   // GBK_TO_UNICODE[32068] := 16#DCDB;
   // GBK_TO_UNICODE[32069] := 16#82D2;
   // GBK_TO_UNICODE[32070] := 16#DCDC;
   // GBK_TO_UNICODE[32071] := 16#82D8;
   // GBK_TO_UNICODE[32072] := 16#DCDD;
   // GBK_TO_UNICODE[32073] := 16#830C;
   // GBK_TO_UNICODE[32074] := 16#DCDE;
   // GBK_TO_UNICODE[32075] := 16#82FB;
   // GBK_TO_UNICODE[32076] := 16#DCDF;
   // GBK_TO_UNICODE[32077] := 16#82D3;
   // GBK_TO_UNICODE[32078] := 16#DCE0;
   // GBK_TO_UNICODE[32079] := 16#8311;
   // GBK_TO_UNICODE[32080] := 16#DCE1;
   // GBK_TO_UNICODE[32081] := 16#831A;
   // GBK_TO_UNICODE[32082] := 16#DCE2;
   // GBK_TO_UNICODE[32083] := 16#8306;
   // GBK_TO_UNICODE[32084] := 16#DCE3;
   // GBK_TO_UNICODE[32085] := 16#8314;
   // GBK_TO_UNICODE[32086] := 16#DCE4;
   // GBK_TO_UNICODE[32087] := 16#8315;
   // GBK_TO_UNICODE[32088] := 16#DCE5;
   // GBK_TO_UNICODE[32089] := 16#82E0;
   // GBK_TO_UNICODE[32090] := 16#DCE6;
   // GBK_TO_UNICODE[32091] := 16#82D5;
   // GBK_TO_UNICODE[32092] := 16#DCE7;
   // GBK_TO_UNICODE[32093] := 16#831C;
   // GBK_TO_UNICODE[32094] := 16#DCE8;
   // GBK_TO_UNICODE[32095] := 16#8351;
   // GBK_TO_UNICODE[32096] := 16#DCE9;
   // GBK_TO_UNICODE[32097] := 16#835B;
   // GBK_TO_UNICODE[32098] := 16#DCEA;
   // GBK_TO_UNICODE[32099] := 16#835C;
   // GBK_TO_UNICODE[32100] := 16#DCEB;
   // GBK_TO_UNICODE[32101] := 16#8308;
   // GBK_TO_UNICODE[32102] := 16#DCEC;
   // GBK_TO_UNICODE[32103] := 16#8392;
   // GBK_TO_UNICODE[32104] := 16#DCED;
   // GBK_TO_UNICODE[32105] := 16#833C;
   // GBK_TO_UNICODE[32106] := 16#DCEE;
   // GBK_TO_UNICODE[32107] := 16#8334;
   // GBK_TO_UNICODE[32108] := 16#DCEF;
   // GBK_TO_UNICODE[32109] := 16#8331;
   // GBK_TO_UNICODE[32110] := 16#DCF0;
   // GBK_TO_UNICODE[32111] := 16#839B;
   // GBK_TO_UNICODE[32112] := 16#DCF1;
   // GBK_TO_UNICODE[32113] := 16#835E;
   // GBK_TO_UNICODE[32114] := 16#DCF2;
   // GBK_TO_UNICODE[32115] := 16#832F;
   // GBK_TO_UNICODE[32116] := 16#DCF3;
   // GBK_TO_UNICODE[32117] := 16#834F;
   // GBK_TO_UNICODE[32118] := 16#DCF4;
   // GBK_TO_UNICODE[32119] := 16#8347;
   // GBK_TO_UNICODE[32120] := 16#DCF5;
   // GBK_TO_UNICODE[32121] := 16#8343;
   // GBK_TO_UNICODE[32122] := 16#DCF6;
   // GBK_TO_UNICODE[32123] := 16#835F;
   // GBK_TO_UNICODE[32124] := 16#DCF7;
   // GBK_TO_UNICODE[32125] := 16#8340;
   // GBK_TO_UNICODE[32126] := 16#DCF8;
   // GBK_TO_UNICODE[32127] := 16#8317;
   // GBK_TO_UNICODE[32128] := 16#DCF9;
   // GBK_TO_UNICODE[32129] := 16#8360;
   // GBK_TO_UNICODE[32130] := 16#DCFA;
   // GBK_TO_UNICODE[32131] := 16#832D;
   // GBK_TO_UNICODE[32132] := 16#DCFB;
   // GBK_TO_UNICODE[32133] := 16#833A;
   // GBK_TO_UNICODE[32134] := 16#DCFC;
   // GBK_TO_UNICODE[32135] := 16#8333;
   // GBK_TO_UNICODE[32136] := 16#DCFD;
   // GBK_TO_UNICODE[32137] := 16#8366;
   // GBK_TO_UNICODE[32138] := 16#DCFE;
   // GBK_TO_UNICODE[32139] := 16#8365;
   // GBK_TO_UNICODE[32140] := 16#DD40;
   // GBK_TO_UNICODE[32141] := 16#8EE5;
   // GBK_TO_UNICODE[32142] := 16#DD41;
   // GBK_TO_UNICODE[32143] := 16#8EE6;
   // GBK_TO_UNICODE[32144] := 16#DD42;
   // GBK_TO_UNICODE[32145] := 16#8EE7;
   // GBK_TO_UNICODE[32146] := 16#DD43;
   // GBK_TO_UNICODE[32147] := 16#8EE8;
   // GBK_TO_UNICODE[32148] := 16#DD44;
   // GBK_TO_UNICODE[32149] := 16#8EE9;
   // GBK_TO_UNICODE[32150] := 16#DD45;
   // GBK_TO_UNICODE[32151] := 16#8EEA;
   // GBK_TO_UNICODE[32152] := 16#DD46;
   // GBK_TO_UNICODE[32153] := 16#8EEB;
   // GBK_TO_UNICODE[32154] := 16#DD47;
   // GBK_TO_UNICODE[32155] := 16#8EEC;
   // GBK_TO_UNICODE[32156] := 16#DD48;
   // GBK_TO_UNICODE[32157] := 16#8EED;
   // GBK_TO_UNICODE[32158] := 16#DD49;
   // GBK_TO_UNICODE[32159] := 16#8EEE;
   // GBK_TO_UNICODE[32160] := 16#DD4A;
   // GBK_TO_UNICODE[32161] := 16#8EEF;
   // GBK_TO_UNICODE[32162] := 16#DD4B;
   // GBK_TO_UNICODE[32163] := 16#8EF0;
   // GBK_TO_UNICODE[32164] := 16#DD4C;
   // GBK_TO_UNICODE[32165] := 16#8EF1;
   // GBK_TO_UNICODE[32166] := 16#DD4D;
   // GBK_TO_UNICODE[32167] := 16#8EF2;
   // GBK_TO_UNICODE[32168] := 16#DD4E;
   // GBK_TO_UNICODE[32169] := 16#8EF3;
   // GBK_TO_UNICODE[32170] := 16#DD4F;
   // GBK_TO_UNICODE[32171] := 16#8EF4;
   // GBK_TO_UNICODE[32172] := 16#DD50;
   // GBK_TO_UNICODE[32173] := 16#8EF5;
   // GBK_TO_UNICODE[32174] := 16#DD51;
   // GBK_TO_UNICODE[32175] := 16#8EF6;
   // GBK_TO_UNICODE[32176] := 16#DD52;
   // GBK_TO_UNICODE[32177] := 16#8EF7;
   // GBK_TO_UNICODE[32178] := 16#DD53;
   // GBK_TO_UNICODE[32179] := 16#8EF8;
   // GBK_TO_UNICODE[32180] := 16#DD54;
   // GBK_TO_UNICODE[32181] := 16#8EF9;
   // GBK_TO_UNICODE[32182] := 16#DD55;
   // GBK_TO_UNICODE[32183] := 16#8EFA;
   // GBK_TO_UNICODE[32184] := 16#DD56;
   // GBK_TO_UNICODE[32185] := 16#8EFB;
   // GBK_TO_UNICODE[32186] := 16#DD57;
   // GBK_TO_UNICODE[32187] := 16#8EFC;
   // GBK_TO_UNICODE[32188] := 16#DD58;
   // GBK_TO_UNICODE[32189] := 16#8EFD;
   // GBK_TO_UNICODE[32190] := 16#DD59;
   // GBK_TO_UNICODE[32191] := 16#8EFE;
   // GBK_TO_UNICODE[32192] := 16#DD5A;
   // GBK_TO_UNICODE[32193] := 16#8EFF;
   // GBK_TO_UNICODE[32194] := 16#DD5B;
   // GBK_TO_UNICODE[32195] := 16#8F00;
   // GBK_TO_UNICODE[32196] := 16#DD5C;
   // GBK_TO_UNICODE[32197] := 16#8F01;
   // GBK_TO_UNICODE[32198] := 16#DD5D;
   // GBK_TO_UNICODE[32199] := 16#8F02;
   // GBK_TO_UNICODE[32200] := 16#DD5E;
   // GBK_TO_UNICODE[32201] := 16#8F03;
   // GBK_TO_UNICODE[32202] := 16#DD5F;
   // GBK_TO_UNICODE[32203] := 16#8F04;
   // GBK_TO_UNICODE[32204] := 16#DD60;
   // GBK_TO_UNICODE[32205] := 16#8F05;
   // GBK_TO_UNICODE[32206] := 16#DD61;
   // GBK_TO_UNICODE[32207] := 16#8F06;
   // GBK_TO_UNICODE[32208] := 16#DD62;
   // GBK_TO_UNICODE[32209] := 16#8F07;
   // GBK_TO_UNICODE[32210] := 16#DD63;
   // GBK_TO_UNICODE[32211] := 16#8F08;
   // GBK_TO_UNICODE[32212] := 16#DD64;
   // GBK_TO_UNICODE[32213] := 16#8F09;
   // GBK_TO_UNICODE[32214] := 16#DD65;
   // GBK_TO_UNICODE[32215] := 16#8F0A;
   // GBK_TO_UNICODE[32216] := 16#DD66;
   // GBK_TO_UNICODE[32217] := 16#8F0B;
   // GBK_TO_UNICODE[32218] := 16#DD67;
   // GBK_TO_UNICODE[32219] := 16#8F0C;
   // GBK_TO_UNICODE[32220] := 16#DD68;
   // GBK_TO_UNICODE[32221] := 16#8F0D;
   // GBK_TO_UNICODE[32222] := 16#DD69;
   // GBK_TO_UNICODE[32223] := 16#8F0E;
   // GBK_TO_UNICODE[32224] := 16#DD6A;
   // GBK_TO_UNICODE[32225] := 16#8F0F;
   // GBK_TO_UNICODE[32226] := 16#DD6B;
   // GBK_TO_UNICODE[32227] := 16#8F10;
   // GBK_TO_UNICODE[32228] := 16#DD6C;
   // GBK_TO_UNICODE[32229] := 16#8F11;
   // GBK_TO_UNICODE[32230] := 16#DD6D;
   // GBK_TO_UNICODE[32231] := 16#8F12;
   // GBK_TO_UNICODE[32232] := 16#DD6E;
   // GBK_TO_UNICODE[32233] := 16#8F13;
   // GBK_TO_UNICODE[32234] := 16#DD6F;
   // GBK_TO_UNICODE[32235] := 16#8F14;
   // GBK_TO_UNICODE[32236] := 16#DD70;
   // GBK_TO_UNICODE[32237] := 16#8F15;
   // GBK_TO_UNICODE[32238] := 16#DD71;
   // GBK_TO_UNICODE[32239] := 16#8F16;
   // GBK_TO_UNICODE[32240] := 16#DD72;
   // GBK_TO_UNICODE[32241] := 16#8F17;
   // GBK_TO_UNICODE[32242] := 16#DD73;
   // GBK_TO_UNICODE[32243] := 16#8F18;
   // GBK_TO_UNICODE[32244] := 16#DD74;
   // GBK_TO_UNICODE[32245] := 16#8F19;
   // GBK_TO_UNICODE[32246] := 16#DD75;
   // GBK_TO_UNICODE[32247] := 16#8F1A;
   // GBK_TO_UNICODE[32248] := 16#DD76;
   // GBK_TO_UNICODE[32249] := 16#8F1B;
   // GBK_TO_UNICODE[32250] := 16#DD77;
   // GBK_TO_UNICODE[32251] := 16#8F1C;
   // GBK_TO_UNICODE[32252] := 16#DD78;
   // GBK_TO_UNICODE[32253] := 16#8F1D;
   // GBK_TO_UNICODE[32254] := 16#DD79;
   // GBK_TO_UNICODE[32255] := 16#8F1E;
   // GBK_TO_UNICODE[32256] := 16#DD7A;
   // GBK_TO_UNICODE[32257] := 16#8F1F;
   // GBK_TO_UNICODE[32258] := 16#DD7B;
   // GBK_TO_UNICODE[32259] := 16#8F20;
   // GBK_TO_UNICODE[32260] := 16#DD7C;
   // GBK_TO_UNICODE[32261] := 16#8F21;
   // GBK_TO_UNICODE[32262] := 16#DD7D;
   // GBK_TO_UNICODE[32263] := 16#8F22;
   // GBK_TO_UNICODE[32264] := 16#DD7E;
   // GBK_TO_UNICODE[32265] := 16#8F23;
   // GBK_TO_UNICODE[32266] := 16#DD80;
   // GBK_TO_UNICODE[32267] := 16#8F24;
   // GBK_TO_UNICODE[32268] := 16#DD81;
   // GBK_TO_UNICODE[32269] := 16#8F25;
   // GBK_TO_UNICODE[32270] := 16#DD82;
   // GBK_TO_UNICODE[32271] := 16#8F26;
   // GBK_TO_UNICODE[32272] := 16#DD83;
   // GBK_TO_UNICODE[32273] := 16#8F27;
   // GBK_TO_UNICODE[32274] := 16#DD84;
   // GBK_TO_UNICODE[32275] := 16#8F28;
   // GBK_TO_UNICODE[32276] := 16#DD85;
   // GBK_TO_UNICODE[32277] := 16#8F29;
   // GBK_TO_UNICODE[32278] := 16#DD86;
   // GBK_TO_UNICODE[32279] := 16#8F2A;
   // GBK_TO_UNICODE[32280] := 16#DD87;
   // GBK_TO_UNICODE[32281] := 16#8F2B;
   // GBK_TO_UNICODE[32282] := 16#DD88;
   // GBK_TO_UNICODE[32283] := 16#8F2C;
   // GBK_TO_UNICODE[32284] := 16#DD89;
   // GBK_TO_UNICODE[32285] := 16#8F2D;
   // GBK_TO_UNICODE[32286] := 16#DD8A;
   // GBK_TO_UNICODE[32287] := 16#8F2E;
   // GBK_TO_UNICODE[32288] := 16#DD8B;
   // GBK_TO_UNICODE[32289] := 16#8F2F;
   // GBK_TO_UNICODE[32290] := 16#DD8C;
   // GBK_TO_UNICODE[32291] := 16#8F30;
   // GBK_TO_UNICODE[32292] := 16#DD8D;
   // GBK_TO_UNICODE[32293] := 16#8F31;
   // GBK_TO_UNICODE[32294] := 16#DD8E;
   // GBK_TO_UNICODE[32295] := 16#8F32;
   // GBK_TO_UNICODE[32296] := 16#DD8F;
   // GBK_TO_UNICODE[32297] := 16#8F33;
   // GBK_TO_UNICODE[32298] := 16#DD90;
   // GBK_TO_UNICODE[32299] := 16#8F34;
   // GBK_TO_UNICODE[32300] := 16#DD91;
   // GBK_TO_UNICODE[32301] := 16#8F35;
   // GBK_TO_UNICODE[32302] := 16#DD92;
   // GBK_TO_UNICODE[32303] := 16#8F36;
   // GBK_TO_UNICODE[32304] := 16#DD93;
   // GBK_TO_UNICODE[32305] := 16#8F37;
   // GBK_TO_UNICODE[32306] := 16#DD94;
   // GBK_TO_UNICODE[32307] := 16#8F38;
   // GBK_TO_UNICODE[32308] := 16#DD95;
   // GBK_TO_UNICODE[32309] := 16#8F39;
   // GBK_TO_UNICODE[32310] := 16#DD96;
   // GBK_TO_UNICODE[32311] := 16#8F3A;
   // GBK_TO_UNICODE[32312] := 16#DD97;
   // GBK_TO_UNICODE[32313] := 16#8F3B;
   // GBK_TO_UNICODE[32314] := 16#DD98;
   // GBK_TO_UNICODE[32315] := 16#8F3C;
   // GBK_TO_UNICODE[32316] := 16#DD99;
   // GBK_TO_UNICODE[32317] := 16#8F3D;
   // GBK_TO_UNICODE[32318] := 16#DD9A;
   // GBK_TO_UNICODE[32319] := 16#8F3E;
   // GBK_TO_UNICODE[32320] := 16#DD9B;
   // GBK_TO_UNICODE[32321] := 16#8F3F;
   // GBK_TO_UNICODE[32322] := 16#DD9C;
   // GBK_TO_UNICODE[32323] := 16#8F40;
   // GBK_TO_UNICODE[32324] := 16#DD9D;
   // GBK_TO_UNICODE[32325] := 16#8F41;
   // GBK_TO_UNICODE[32326] := 16#DD9E;
   // GBK_TO_UNICODE[32327] := 16#8F42;
   // GBK_TO_UNICODE[32328] := 16#DD9F;
   // GBK_TO_UNICODE[32329] := 16#8F43;
   // GBK_TO_UNICODE[32330] := 16#DDA0;
   // GBK_TO_UNICODE[32331] := 16#8F44;
   // GBK_TO_UNICODE[32332] := 16#DDA1;
   // GBK_TO_UNICODE[32333] := 16#8368;
   // GBK_TO_UNICODE[32334] := 16#DDA2;
   // GBK_TO_UNICODE[32335] := 16#831B;
   // GBK_TO_UNICODE[32336] := 16#DDA3;
   // GBK_TO_UNICODE[32337] := 16#8369;
   // GBK_TO_UNICODE[32338] := 16#DDA4;
   // GBK_TO_UNICODE[32339] := 16#836C;
   // GBK_TO_UNICODE[32340] := 16#DDA5;
   // GBK_TO_UNICODE[32341] := 16#836A;
   // GBK_TO_UNICODE[32342] := 16#DDA6;
   // GBK_TO_UNICODE[32343] := 16#836D;
   // GBK_TO_UNICODE[32344] := 16#DDA7;
   // GBK_TO_UNICODE[32345] := 16#836E;
   // GBK_TO_UNICODE[32346] := 16#DDA8;
   // GBK_TO_UNICODE[32347] := 16#83B0;
   // GBK_TO_UNICODE[32348] := 16#DDA9;
   // GBK_TO_UNICODE[32349] := 16#8378;
   // GBK_TO_UNICODE[32350] := 16#DDAA;
   // GBK_TO_UNICODE[32351] := 16#83B3;
   // GBK_TO_UNICODE[32352] := 16#DDAB;
   // GBK_TO_UNICODE[32353] := 16#83B4;
   // GBK_TO_UNICODE[32354] := 16#DDAC;
   // GBK_TO_UNICODE[32355] := 16#83A0;
   // GBK_TO_UNICODE[32356] := 16#DDAD;
   // GBK_TO_UNICODE[32357] := 16#83AA;
   // GBK_TO_UNICODE[32358] := 16#DDAE;
   // GBK_TO_UNICODE[32359] := 16#8393;
   // GBK_TO_UNICODE[32360] := 16#DDAF;
   // GBK_TO_UNICODE[32361] := 16#839C;
   // GBK_TO_UNICODE[32362] := 16#DDB0;
   // GBK_TO_UNICODE[32363] := 16#8385;
   // GBK_TO_UNICODE[32364] := 16#DDB1;
   // GBK_TO_UNICODE[32365] := 16#837C;
   // GBK_TO_UNICODE[32366] := 16#DDB2;
   // GBK_TO_UNICODE[32367] := 16#83B6;
   // GBK_TO_UNICODE[32368] := 16#DDB3;
   // GBK_TO_UNICODE[32369] := 16#83A9;
   // GBK_TO_UNICODE[32370] := 16#DDB4;
   // GBK_TO_UNICODE[32371] := 16#837D;
   // GBK_TO_UNICODE[32372] := 16#DDB5;
   // GBK_TO_UNICODE[32373] := 16#83B8;
   // GBK_TO_UNICODE[32374] := 16#DDB6;
   // GBK_TO_UNICODE[32375] := 16#837B;
   // GBK_TO_UNICODE[32376] := 16#DDB7;
   // GBK_TO_UNICODE[32377] := 16#8398;
   // GBK_TO_UNICODE[32378] := 16#DDB8;
   // GBK_TO_UNICODE[32379] := 16#839E;
   // GBK_TO_UNICODE[32380] := 16#DDB9;
   // GBK_TO_UNICODE[32381] := 16#83A8;
   // GBK_TO_UNICODE[32382] := 16#DDBA;
   // GBK_TO_UNICODE[32383] := 16#83BA;
   // GBK_TO_UNICODE[32384] := 16#DDBB;
   // GBK_TO_UNICODE[32385] := 16#83BC;
   // GBK_TO_UNICODE[32386] := 16#DDBC;
   // GBK_TO_UNICODE[32387] := 16#83C1;
   // GBK_TO_UNICODE[32388] := 16#DDBD;
   // GBK_TO_UNICODE[32389] := 16#8401;
   // GBK_TO_UNICODE[32390] := 16#DDBE;
   // GBK_TO_UNICODE[32391] := 16#83E5;
   // GBK_TO_UNICODE[32392] := 16#DDBF;
   // GBK_TO_UNICODE[32393] := 16#83D8;
   // GBK_TO_UNICODE[32394] := 16#DDC0;
   // GBK_TO_UNICODE[32395] := 16#5807;
   // GBK_TO_UNICODE[32396] := 16#DDC1;
   // GBK_TO_UNICODE[32397] := 16#8418;
   // GBK_TO_UNICODE[32398] := 16#DDC2;
   // GBK_TO_UNICODE[32399] := 16#840B;
   // GBK_TO_UNICODE[32400] := 16#DDC3;
   // GBK_TO_UNICODE[32401] := 16#83DD;
   // GBK_TO_UNICODE[32402] := 16#DDC4;
   // GBK_TO_UNICODE[32403] := 16#83FD;
   // GBK_TO_UNICODE[32404] := 16#DDC5;
   // GBK_TO_UNICODE[32405] := 16#83D6;
   // GBK_TO_UNICODE[32406] := 16#DDC6;
   // GBK_TO_UNICODE[32407] := 16#841C;
   // GBK_TO_UNICODE[32408] := 16#DDC7;
   // GBK_TO_UNICODE[32409] := 16#8438;
   // GBK_TO_UNICODE[32410] := 16#DDC8;
   // GBK_TO_UNICODE[32411] := 16#8411;
   // GBK_TO_UNICODE[32412] := 16#DDC9;
   // GBK_TO_UNICODE[32413] := 16#8406;
   // GBK_TO_UNICODE[32414] := 16#DDCA;
   // GBK_TO_UNICODE[32415] := 16#83D4;
   // GBK_TO_UNICODE[32416] := 16#DDCB;
   // GBK_TO_UNICODE[32417] := 16#83DF;
   // GBK_TO_UNICODE[32418] := 16#DDCC;
   // GBK_TO_UNICODE[32419] := 16#840F;
   // GBK_TO_UNICODE[32420] := 16#DDCD;
   // GBK_TO_UNICODE[32421] := 16#8403;
   // GBK_TO_UNICODE[32422] := 16#DDCE;
   // GBK_TO_UNICODE[32423] := 16#83F8;
   // GBK_TO_UNICODE[32424] := 16#DDCF;
   // GBK_TO_UNICODE[32425] := 16#83F9;
   // GBK_TO_UNICODE[32426] := 16#DDD0;
   // GBK_TO_UNICODE[32427] := 16#83EA;
   // GBK_TO_UNICODE[32428] := 16#DDD1;
   // GBK_TO_UNICODE[32429] := 16#83C5;
   // GBK_TO_UNICODE[32430] := 16#DDD2;
   // GBK_TO_UNICODE[32431] := 16#83C0;
   // GBK_TO_UNICODE[32432] := 16#DDD3;
   // GBK_TO_UNICODE[32433] := 16#8426;
   // GBK_TO_UNICODE[32434] := 16#DDD4;
   // GBK_TO_UNICODE[32435] := 16#83F0;
   // GBK_TO_UNICODE[32436] := 16#DDD5;
   // GBK_TO_UNICODE[32437] := 16#83E1;
   // GBK_TO_UNICODE[32438] := 16#DDD6;
   // GBK_TO_UNICODE[32439] := 16#845C;
   // GBK_TO_UNICODE[32440] := 16#DDD7;
   // GBK_TO_UNICODE[32441] := 16#8451;
   // GBK_TO_UNICODE[32442] := 16#DDD8;
   // GBK_TO_UNICODE[32443] := 16#845A;
   // GBK_TO_UNICODE[32444] := 16#DDD9;
   // GBK_TO_UNICODE[32445] := 16#8459;
   // GBK_TO_UNICODE[32446] := 16#DDDA;
   // GBK_TO_UNICODE[32447] := 16#8473;
   // GBK_TO_UNICODE[32448] := 16#DDDB;
   // GBK_TO_UNICODE[32449] := 16#8487;
   // GBK_TO_UNICODE[32450] := 16#DDDC;
   // GBK_TO_UNICODE[32451] := 16#8488;
   // GBK_TO_UNICODE[32452] := 16#DDDD;
   // GBK_TO_UNICODE[32453] := 16#847A;
   // GBK_TO_UNICODE[32454] := 16#DDDE;
   // GBK_TO_UNICODE[32455] := 16#8489;
   // GBK_TO_UNICODE[32456] := 16#DDDF;
   // GBK_TO_UNICODE[32457] := 16#8478;
   // GBK_TO_UNICODE[32458] := 16#DDE0;
   // GBK_TO_UNICODE[32459] := 16#843C;
   // GBK_TO_UNICODE[32460] := 16#DDE1;
   // GBK_TO_UNICODE[32461] := 16#8446;
   // GBK_TO_UNICODE[32462] := 16#DDE2;
   // GBK_TO_UNICODE[32463] := 16#8469;
   // GBK_TO_UNICODE[32464] := 16#DDE3;
   // GBK_TO_UNICODE[32465] := 16#8476;
   // GBK_TO_UNICODE[32466] := 16#DDE4;
   // GBK_TO_UNICODE[32467] := 16#848C;
   // GBK_TO_UNICODE[32468] := 16#DDE5;
   // GBK_TO_UNICODE[32469] := 16#848E;
   // GBK_TO_UNICODE[32470] := 16#DDE6;
   // GBK_TO_UNICODE[32471] := 16#8431;
   // GBK_TO_UNICODE[32472] := 16#DDE7;
   // GBK_TO_UNICODE[32473] := 16#846D;
   // GBK_TO_UNICODE[32474] := 16#DDE8;
   // GBK_TO_UNICODE[32475] := 16#84C1;
   // GBK_TO_UNICODE[32476] := 16#DDE9;
   // GBK_TO_UNICODE[32477] := 16#84CD;
   // GBK_TO_UNICODE[32478] := 16#DDEA;
   // GBK_TO_UNICODE[32479] := 16#84D0;
   // GBK_TO_UNICODE[32480] := 16#DDEB;
   // GBK_TO_UNICODE[32481] := 16#84E6;
   // GBK_TO_UNICODE[32482] := 16#DDEC;
   // GBK_TO_UNICODE[32483] := 16#84BD;
   // GBK_TO_UNICODE[32484] := 16#DDED;
   // GBK_TO_UNICODE[32485] := 16#84D3;
   // GBK_TO_UNICODE[32486] := 16#DDEE;
   // GBK_TO_UNICODE[32487] := 16#84CA;
   // GBK_TO_UNICODE[32488] := 16#DDEF;
   // GBK_TO_UNICODE[32489] := 16#84BF;
   // GBK_TO_UNICODE[32490] := 16#DDF0;
   // GBK_TO_UNICODE[32491] := 16#84BA;
   // GBK_TO_UNICODE[32492] := 16#DDF1;
   // GBK_TO_UNICODE[32493] := 16#84E0;
   // GBK_TO_UNICODE[32494] := 16#DDF2;
   // GBK_TO_UNICODE[32495] := 16#84A1;
   // GBK_TO_UNICODE[32496] := 16#DDF3;
   // GBK_TO_UNICODE[32497] := 16#84B9;
   // GBK_TO_UNICODE[32498] := 16#DDF4;
   // GBK_TO_UNICODE[32499] := 16#84B4;
   // GBK_TO_UNICODE[32500] := 16#DDF5;
   // GBK_TO_UNICODE[32501] := 16#8497;
   // GBK_TO_UNICODE[32502] := 16#DDF6;
   // GBK_TO_UNICODE[32503] := 16#84E5;
   // GBK_TO_UNICODE[32504] := 16#DDF7;
   // GBK_TO_UNICODE[32505] := 16#84E3;
   // GBK_TO_UNICODE[32506] := 16#DDF8;
   // GBK_TO_UNICODE[32507] := 16#850C;
   // GBK_TO_UNICODE[32508] := 16#DDF9;
   // GBK_TO_UNICODE[32509] := 16#750D;
   // GBK_TO_UNICODE[32510] := 16#DDFA;
   // GBK_TO_UNICODE[32511] := 16#8538;
   // GBK_TO_UNICODE[32512] := 16#DDFB;
   // GBK_TO_UNICODE[32513] := 16#84F0;
   // GBK_TO_UNICODE[32514] := 16#DDFC;
   // GBK_TO_UNICODE[32515] := 16#8539;
   // GBK_TO_UNICODE[32516] := 16#DDFD;
   // GBK_TO_UNICODE[32517] := 16#851F;
   // GBK_TO_UNICODE[32518] := 16#DDFE;
   // GBK_TO_UNICODE[32519] := 16#853A;
   // GBK_TO_UNICODE[32520] := 16#DE40;
   // GBK_TO_UNICODE[32521] := 16#8F45;
   // GBK_TO_UNICODE[32522] := 16#DE41;
   // GBK_TO_UNICODE[32523] := 16#8F46;
   // GBK_TO_UNICODE[32524] := 16#DE42;
   // GBK_TO_UNICODE[32525] := 16#8F47;
   // GBK_TO_UNICODE[32526] := 16#DE43;
   // GBK_TO_UNICODE[32527] := 16#8F48;
   // GBK_TO_UNICODE[32528] := 16#DE44;
   // GBK_TO_UNICODE[32529] := 16#8F49;
   // GBK_TO_UNICODE[32530] := 16#DE45;
   // GBK_TO_UNICODE[32531] := 16#8F4A;
   // GBK_TO_UNICODE[32532] := 16#DE46;
   // GBK_TO_UNICODE[32533] := 16#8F4B;
   // GBK_TO_UNICODE[32534] := 16#DE47;
   // GBK_TO_UNICODE[32535] := 16#8F4C;
   // GBK_TO_UNICODE[32536] := 16#DE48;
   // GBK_TO_UNICODE[32537] := 16#8F4D;
   // GBK_TO_UNICODE[32538] := 16#DE49;
   // GBK_TO_UNICODE[32539] := 16#8F4E;
   // GBK_TO_UNICODE[32540] := 16#DE4A;
   // GBK_TO_UNICODE[32541] := 16#8F4F;
   // GBK_TO_UNICODE[32542] := 16#DE4B;
   // GBK_TO_UNICODE[32543] := 16#8F50;
   // GBK_TO_UNICODE[32544] := 16#DE4C;
   // GBK_TO_UNICODE[32545] := 16#8F51;
   // GBK_TO_UNICODE[32546] := 16#DE4D;
   // GBK_TO_UNICODE[32547] := 16#8F52;
   // GBK_TO_UNICODE[32548] := 16#DE4E;
   // GBK_TO_UNICODE[32549] := 16#8F53;
   // GBK_TO_UNICODE[32550] := 16#DE4F;
   // GBK_TO_UNICODE[32551] := 16#8F54;
   // GBK_TO_UNICODE[32552] := 16#DE50;
   // GBK_TO_UNICODE[32553] := 16#8F55;
   // GBK_TO_UNICODE[32554] := 16#DE51;
   // GBK_TO_UNICODE[32555] := 16#8F56;
   // GBK_TO_UNICODE[32556] := 16#DE52;
   // GBK_TO_UNICODE[32557] := 16#8F57;
   // GBK_TO_UNICODE[32558] := 16#DE53;
   // GBK_TO_UNICODE[32559] := 16#8F58;
   // GBK_TO_UNICODE[32560] := 16#DE54;
   // GBK_TO_UNICODE[32561] := 16#8F59;
   // GBK_TO_UNICODE[32562] := 16#DE55;
   // GBK_TO_UNICODE[32563] := 16#8F5A;
   // GBK_TO_UNICODE[32564] := 16#DE56;
   // GBK_TO_UNICODE[32565] := 16#8F5B;
   // GBK_TO_UNICODE[32566] := 16#DE57;
   // GBK_TO_UNICODE[32567] := 16#8F5C;
   // GBK_TO_UNICODE[32568] := 16#DE58;
   // GBK_TO_UNICODE[32569] := 16#8F5D;
   // GBK_TO_UNICODE[32570] := 16#DE59;
   // GBK_TO_UNICODE[32571] := 16#8F5E;
   // GBK_TO_UNICODE[32572] := 16#DE5A;
   // GBK_TO_UNICODE[32573] := 16#8F5F;
   // GBK_TO_UNICODE[32574] := 16#DE5B;
   // GBK_TO_UNICODE[32575] := 16#8F60;
   // GBK_TO_UNICODE[32576] := 16#DE5C;
   // GBK_TO_UNICODE[32577] := 16#8F61;
   // GBK_TO_UNICODE[32578] := 16#DE5D;
   // GBK_TO_UNICODE[32579] := 16#8F62;
   // GBK_TO_UNICODE[32580] := 16#DE5E;
   // GBK_TO_UNICODE[32581] := 16#8F63;
   // GBK_TO_UNICODE[32582] := 16#DE5F;
   // GBK_TO_UNICODE[32583] := 16#8F64;
   // GBK_TO_UNICODE[32584] := 16#DE60;
   // GBK_TO_UNICODE[32585] := 16#8F65;
   // GBK_TO_UNICODE[32586] := 16#DE61;
   // GBK_TO_UNICODE[32587] := 16#8F6A;
   // GBK_TO_UNICODE[32588] := 16#DE62;
   // GBK_TO_UNICODE[32589] := 16#8F80;
   // GBK_TO_UNICODE[32590] := 16#DE63;
   // GBK_TO_UNICODE[32591] := 16#8F8C;
   // GBK_TO_UNICODE[32592] := 16#DE64;
   // GBK_TO_UNICODE[32593] := 16#8F92;
   // GBK_TO_UNICODE[32594] := 16#DE65;
   // GBK_TO_UNICODE[32595] := 16#8F9D;
   // GBK_TO_UNICODE[32596] := 16#DE66;
   // GBK_TO_UNICODE[32597] := 16#8FA0;
   // GBK_TO_UNICODE[32598] := 16#DE67;
   // GBK_TO_UNICODE[32599] := 16#8FA1;
   // GBK_TO_UNICODE[32600] := 16#DE68;
   // GBK_TO_UNICODE[32601] := 16#8FA2;
   // GBK_TO_UNICODE[32602] := 16#DE69;
   // GBK_TO_UNICODE[32603] := 16#8FA4;
   // GBK_TO_UNICODE[32604] := 16#DE6A;
   // GBK_TO_UNICODE[32605] := 16#8FA5;
   // GBK_TO_UNICODE[32606] := 16#DE6B;
   // GBK_TO_UNICODE[32607] := 16#8FA6;
   // GBK_TO_UNICODE[32608] := 16#DE6C;
   // GBK_TO_UNICODE[32609] := 16#8FA7;
   // GBK_TO_UNICODE[32610] := 16#DE6D;
   // GBK_TO_UNICODE[32611] := 16#8FAA;
   // GBK_TO_UNICODE[32612] := 16#DE6E;
   // GBK_TO_UNICODE[32613] := 16#8FAC;
   // GBK_TO_UNICODE[32614] := 16#DE6F;
   // GBK_TO_UNICODE[32615] := 16#8FAD;
   // GBK_TO_UNICODE[32616] := 16#DE70;
   // GBK_TO_UNICODE[32617] := 16#8FAE;
   // GBK_TO_UNICODE[32618] := 16#DE71;
   // GBK_TO_UNICODE[32619] := 16#8FAF;
   // GBK_TO_UNICODE[32620] := 16#DE72;
   // GBK_TO_UNICODE[32621] := 16#8FB2;
   // GBK_TO_UNICODE[32622] := 16#DE73;
   // GBK_TO_UNICODE[32623] := 16#8FB3;
   // GBK_TO_UNICODE[32624] := 16#DE74;
   // GBK_TO_UNICODE[32625] := 16#8FB4;
   // GBK_TO_UNICODE[32626] := 16#DE75;
   // GBK_TO_UNICODE[32627] := 16#8FB5;
   // GBK_TO_UNICODE[32628] := 16#DE76;
   // GBK_TO_UNICODE[32629] := 16#8FB7;
   // GBK_TO_UNICODE[32630] := 16#DE77;
   // GBK_TO_UNICODE[32631] := 16#8FB8;
   // GBK_TO_UNICODE[32632] := 16#DE78;
   // GBK_TO_UNICODE[32633] := 16#8FBA;
   // GBK_TO_UNICODE[32634] := 16#DE79;
   // GBK_TO_UNICODE[32635] := 16#8FBB;
   // GBK_TO_UNICODE[32636] := 16#DE7A;
   // GBK_TO_UNICODE[32637] := 16#8FBC;
   // GBK_TO_UNICODE[32638] := 16#DE7B;
   // GBK_TO_UNICODE[32639] := 16#8FBF;
   // GBK_TO_UNICODE[32640] := 16#DE7C;
   // GBK_TO_UNICODE[32641] := 16#8FC0;
   // GBK_TO_UNICODE[32642] := 16#DE7D;
   // GBK_TO_UNICODE[32643] := 16#8FC3;
   // GBK_TO_UNICODE[32644] := 16#DE7E;
   // GBK_TO_UNICODE[32645] := 16#8FC6;
   // GBK_TO_UNICODE[32646] := 16#DE80;
   // GBK_TO_UNICODE[32647] := 16#8FC9;
   // GBK_TO_UNICODE[32648] := 16#DE81;
   // GBK_TO_UNICODE[32649] := 16#8FCA;
   // GBK_TO_UNICODE[32650] := 16#DE82;
   // GBK_TO_UNICODE[32651] := 16#8FCB;
   // GBK_TO_UNICODE[32652] := 16#DE83;
   // GBK_TO_UNICODE[32653] := 16#8FCC;
   // GBK_TO_UNICODE[32654] := 16#DE84;
   // GBK_TO_UNICODE[32655] := 16#8FCD;
   // GBK_TO_UNICODE[32656] := 16#DE85;
   // GBK_TO_UNICODE[32657] := 16#8FCF;
   // GBK_TO_UNICODE[32658] := 16#DE86;
   // GBK_TO_UNICODE[32659] := 16#8FD2;
   // GBK_TO_UNICODE[32660] := 16#DE87;
   // GBK_TO_UNICODE[32661] := 16#8FD6;
   // GBK_TO_UNICODE[32662] := 16#DE88;
   // GBK_TO_UNICODE[32663] := 16#8FD7;
   // GBK_TO_UNICODE[32664] := 16#DE89;
   // GBK_TO_UNICODE[32665] := 16#8FDA;
   // GBK_TO_UNICODE[32666] := 16#DE8A;
   // GBK_TO_UNICODE[32667] := 16#8FE0;
   // GBK_TO_UNICODE[32668] := 16#DE8B;
   // GBK_TO_UNICODE[32669] := 16#8FE1;
   // GBK_TO_UNICODE[32670] := 16#DE8C;
   // GBK_TO_UNICODE[32671] := 16#8FE3;
   // GBK_TO_UNICODE[32672] := 16#DE8D;
   // GBK_TO_UNICODE[32673] := 16#8FE7;
   // GBK_TO_UNICODE[32674] := 16#DE8E;
   // GBK_TO_UNICODE[32675] := 16#8FEC;
   // GBK_TO_UNICODE[32676] := 16#DE8F;
   // GBK_TO_UNICODE[32677] := 16#8FEF;
   // GBK_TO_UNICODE[32678] := 16#DE90;
   // GBK_TO_UNICODE[32679] := 16#8FF1;
   // GBK_TO_UNICODE[32680] := 16#DE91;
   // GBK_TO_UNICODE[32681] := 16#8FF2;
   // GBK_TO_UNICODE[32682] := 16#DE92;
   // GBK_TO_UNICODE[32683] := 16#8FF4;
   // GBK_TO_UNICODE[32684] := 16#DE93;
   // GBK_TO_UNICODE[32685] := 16#8FF5;
   // GBK_TO_UNICODE[32686] := 16#DE94;
   // GBK_TO_UNICODE[32687] := 16#8FF6;
   // GBK_TO_UNICODE[32688] := 16#DE95;
   // GBK_TO_UNICODE[32689] := 16#8FFA;
   // GBK_TO_UNICODE[32690] := 16#DE96;
   // GBK_TO_UNICODE[32691] := 16#8FFB;
   // GBK_TO_UNICODE[32692] := 16#DE97;
   // GBK_TO_UNICODE[32693] := 16#8FFC;
   // GBK_TO_UNICODE[32694] := 16#DE98;
   // GBK_TO_UNICODE[32695] := 16#8FFE;
   // GBK_TO_UNICODE[32696] := 16#DE99;
   // GBK_TO_UNICODE[32697] := 16#8FFF;
   // GBK_TO_UNICODE[32698] := 16#DE9A;
   // GBK_TO_UNICODE[32699] := 16#9007;
   // GBK_TO_UNICODE[32700] := 16#DE9B;
   // GBK_TO_UNICODE[32701] := 16#9008;
   // GBK_TO_UNICODE[32702] := 16#DE9C;
   // GBK_TO_UNICODE[32703] := 16#900C;
   // GBK_TO_UNICODE[32704] := 16#DE9D;
   // GBK_TO_UNICODE[32705] := 16#900E;
   // GBK_TO_UNICODE[32706] := 16#DE9E;
   // GBK_TO_UNICODE[32707] := 16#9013;
   // GBK_TO_UNICODE[32708] := 16#DE9F;
   // GBK_TO_UNICODE[32709] := 16#9015;
   // GBK_TO_UNICODE[32710] := 16#DEA0;
   // GBK_TO_UNICODE[32711] := 16#9018;
   // GBK_TO_UNICODE[32712] := 16#DEA1;
   // GBK_TO_UNICODE[32713] := 16#8556;
   // GBK_TO_UNICODE[32714] := 16#DEA2;
   // GBK_TO_UNICODE[32715] := 16#853B;
   // GBK_TO_UNICODE[32716] := 16#DEA3;
   // GBK_TO_UNICODE[32717] := 16#84FF;
   // GBK_TO_UNICODE[32718] := 16#DEA4;
   // GBK_TO_UNICODE[32719] := 16#84FC;
   // GBK_TO_UNICODE[32720] := 16#DEA5;
   // GBK_TO_UNICODE[32721] := 16#8559;
   // GBK_TO_UNICODE[32722] := 16#DEA6;
   // GBK_TO_UNICODE[32723] := 16#8548;
   // GBK_TO_UNICODE[32724] := 16#DEA7;
   // GBK_TO_UNICODE[32725] := 16#8568;
   // GBK_TO_UNICODE[32726] := 16#DEA8;
   // GBK_TO_UNICODE[32727] := 16#8564;
   // GBK_TO_UNICODE[32728] := 16#DEA9;
   // GBK_TO_UNICODE[32729] := 16#855E;
   // GBK_TO_UNICODE[32730] := 16#DEAA;
   // GBK_TO_UNICODE[32731] := 16#857A;
   // GBK_TO_UNICODE[32732] := 16#DEAB;
   // GBK_TO_UNICODE[32733] := 16#77A2;
   // GBK_TO_UNICODE[32734] := 16#DEAC;
   // GBK_TO_UNICODE[32735] := 16#8543;
   // GBK_TO_UNICODE[32736] := 16#DEAD;
   // GBK_TO_UNICODE[32737] := 16#8572;
   // GBK_TO_UNICODE[32738] := 16#DEAE;
   // GBK_TO_UNICODE[32739] := 16#857B;
   // GBK_TO_UNICODE[32740] := 16#DEAF;
   // GBK_TO_UNICODE[32741] := 16#85A4;
   // GBK_TO_UNICODE[32742] := 16#DEB0;
   // GBK_TO_UNICODE[32743] := 16#85A8;
   // GBK_TO_UNICODE[32744] := 16#DEB1;
   // GBK_TO_UNICODE[32745] := 16#8587;
   // GBK_TO_UNICODE[32746] := 16#DEB2;
   // GBK_TO_UNICODE[32747] := 16#858F;
   // GBK_TO_UNICODE[32748] := 16#DEB3;
   // GBK_TO_UNICODE[32749] := 16#8579;
   // GBK_TO_UNICODE[32750] := 16#DEB4;
   // GBK_TO_UNICODE[32751] := 16#85AE;
   // GBK_TO_UNICODE[32752] := 16#DEB5;
   // GBK_TO_UNICODE[32753] := 16#859C;
   // GBK_TO_UNICODE[32754] := 16#DEB6;
   // GBK_TO_UNICODE[32755] := 16#8585;
   // GBK_TO_UNICODE[32756] := 16#DEB7;
   // GBK_TO_UNICODE[32757] := 16#85B9;
   // GBK_TO_UNICODE[32758] := 16#DEB8;
   // GBK_TO_UNICODE[32759] := 16#85B7;
   // GBK_TO_UNICODE[32760] := 16#DEB9;
   // GBK_TO_UNICODE[32761] := 16#85B0;
   // GBK_TO_UNICODE[32762] := 16#DEBA;
   // GBK_TO_UNICODE[32763] := 16#85D3;
   // GBK_TO_UNICODE[32764] := 16#DEBB;
   // GBK_TO_UNICODE[32765] := 16#85C1;
   // GBK_TO_UNICODE[32766] := 16#DEBC;
   // GBK_TO_UNICODE[32767] := 16#85DC;
   // GBK_TO_UNICODE[32768] := 16#DEBD;
   // GBK_TO_UNICODE[32769] := 16#85FF;
   // GBK_TO_UNICODE[32770] := 16#DEBE;
   // GBK_TO_UNICODE[32771] := 16#8627;
   // GBK_TO_UNICODE[32772] := 16#DEBF;
   // GBK_TO_UNICODE[32773] := 16#8605;
   // GBK_TO_UNICODE[32774] := 16#DEC0;
   // GBK_TO_UNICODE[32775] := 16#8629;
   // GBK_TO_UNICODE[32776] := 16#DEC1;
   // GBK_TO_UNICODE[32777] := 16#8616;
   // GBK_TO_UNICODE[32778] := 16#DEC2;
   // GBK_TO_UNICODE[32779] := 16#863C;
   // GBK_TO_UNICODE[32780] := 16#DEC3;
   // GBK_TO_UNICODE[32781] := 16#5EFE;
   // GBK_TO_UNICODE[32782] := 16#DEC4;
   // GBK_TO_UNICODE[32783] := 16#5F08;
   // GBK_TO_UNICODE[32784] := 16#DEC5;
   // GBK_TO_UNICODE[32785] := 16#593C;
   // GBK_TO_UNICODE[32786] := 16#DEC6;
   // GBK_TO_UNICODE[32787] := 16#5941;
   // GBK_TO_UNICODE[32788] := 16#DEC7;
   // GBK_TO_UNICODE[32789] := 16#8037;
   // GBK_TO_UNICODE[32790] := 16#DEC8;
   // GBK_TO_UNICODE[32791] := 16#5955;
   // GBK_TO_UNICODE[32792] := 16#DEC9;
   // GBK_TO_UNICODE[32793] := 16#595A;
   // GBK_TO_UNICODE[32794] := 16#DECA;
   // GBK_TO_UNICODE[32795] := 16#5958;
   // GBK_TO_UNICODE[32796] := 16#DECB;
   // GBK_TO_UNICODE[32797] := 16#530F;
   // GBK_TO_UNICODE[32798] := 16#DECC;
   // GBK_TO_UNICODE[32799] := 16#5C22;
   // GBK_TO_UNICODE[32800] := 16#DECD;
   // GBK_TO_UNICODE[32801] := 16#5C25;
   // GBK_TO_UNICODE[32802] := 16#DECE;
   // GBK_TO_UNICODE[32803] := 16#5C2C;
   // GBK_TO_UNICODE[32804] := 16#DECF;
   // GBK_TO_UNICODE[32805] := 16#5C34;
   // GBK_TO_UNICODE[32806] := 16#DED0;
   // GBK_TO_UNICODE[32807] := 16#624C;
   // GBK_TO_UNICODE[32808] := 16#DED1;
   // GBK_TO_UNICODE[32809] := 16#626A;
   // GBK_TO_UNICODE[32810] := 16#DED2;
   // GBK_TO_UNICODE[32811] := 16#629F;
   // GBK_TO_UNICODE[32812] := 16#DED3;
   // GBK_TO_UNICODE[32813] := 16#62BB;
   // GBK_TO_UNICODE[32814] := 16#DED4;
   // GBK_TO_UNICODE[32815] := 16#62CA;
   // GBK_TO_UNICODE[32816] := 16#DED5;
   // GBK_TO_UNICODE[32817] := 16#62DA;
   // GBK_TO_UNICODE[32818] := 16#DED6;
   // GBK_TO_UNICODE[32819] := 16#62D7;
   // GBK_TO_UNICODE[32820] := 16#DED7;
   // GBK_TO_UNICODE[32821] := 16#62EE;
   // GBK_TO_UNICODE[32822] := 16#DED8;
   // GBK_TO_UNICODE[32823] := 16#6322;
   // GBK_TO_UNICODE[32824] := 16#DED9;
   // GBK_TO_UNICODE[32825] := 16#62F6;
   // GBK_TO_UNICODE[32826] := 16#DEDA;
   // GBK_TO_UNICODE[32827] := 16#6339;
   // GBK_TO_UNICODE[32828] := 16#DEDB;
   // GBK_TO_UNICODE[32829] := 16#634B;
   // GBK_TO_UNICODE[32830] := 16#DEDC;
   // GBK_TO_UNICODE[32831] := 16#6343;
   // GBK_TO_UNICODE[32832] := 16#DEDD;
   // GBK_TO_UNICODE[32833] := 16#63AD;
   // GBK_TO_UNICODE[32834] := 16#DEDE;
   // GBK_TO_UNICODE[32835] := 16#63F6;
   // GBK_TO_UNICODE[32836] := 16#DEDF;
   // GBK_TO_UNICODE[32837] := 16#6371;
   // GBK_TO_UNICODE[32838] := 16#DEE0;
   // GBK_TO_UNICODE[32839] := 16#637A;
   // GBK_TO_UNICODE[32840] := 16#DEE1;
   // GBK_TO_UNICODE[32841] := 16#638E;
   // GBK_TO_UNICODE[32842] := 16#DEE2;
   // GBK_TO_UNICODE[32843] := 16#63B4;
   // GBK_TO_UNICODE[32844] := 16#DEE3;
   // GBK_TO_UNICODE[32845] := 16#636D;
   // GBK_TO_UNICODE[32846] := 16#DEE4;
   // GBK_TO_UNICODE[32847] := 16#63AC;
   // GBK_TO_UNICODE[32848] := 16#DEE5;
   // GBK_TO_UNICODE[32849] := 16#638A;
   // GBK_TO_UNICODE[32850] := 16#DEE6;
   // GBK_TO_UNICODE[32851] := 16#6369;
   // GBK_TO_UNICODE[32852] := 16#DEE7;
   // GBK_TO_UNICODE[32853] := 16#63AE;
   // GBK_TO_UNICODE[32854] := 16#DEE8;
   // GBK_TO_UNICODE[32855] := 16#63BC;
   // GBK_TO_UNICODE[32856] := 16#DEE9;
   // GBK_TO_UNICODE[32857] := 16#63F2;
   // GBK_TO_UNICODE[32858] := 16#DEEA;
   // GBK_TO_UNICODE[32859] := 16#63F8;
   // GBK_TO_UNICODE[32860] := 16#DEEB;
   // GBK_TO_UNICODE[32861] := 16#63E0;
   // GBK_TO_UNICODE[32862] := 16#DEEC;
   // GBK_TO_UNICODE[32863] := 16#63FF;
   // GBK_TO_UNICODE[32864] := 16#DEED;
   // GBK_TO_UNICODE[32865] := 16#63C4;
   // GBK_TO_UNICODE[32866] := 16#DEEE;
   // GBK_TO_UNICODE[32867] := 16#63DE;
   // GBK_TO_UNICODE[32868] := 16#DEEF;
   // GBK_TO_UNICODE[32869] := 16#63CE;
   // GBK_TO_UNICODE[32870] := 16#DEF0;
   // GBK_TO_UNICODE[32871] := 16#6452;
   // GBK_TO_UNICODE[32872] := 16#DEF1;
   // GBK_TO_UNICODE[32873] := 16#63C6;
   // GBK_TO_UNICODE[32874] := 16#DEF2;
   // GBK_TO_UNICODE[32875] := 16#63BE;
   // GBK_TO_UNICODE[32876] := 16#DEF3;
   // GBK_TO_UNICODE[32877] := 16#6445;
   // GBK_TO_UNICODE[32878] := 16#DEF4;
   // GBK_TO_UNICODE[32879] := 16#6441;
   // GBK_TO_UNICODE[32880] := 16#DEF5;
   // GBK_TO_UNICODE[32881] := 16#640B;
   // GBK_TO_UNICODE[32882] := 16#DEF6;
   // GBK_TO_UNICODE[32883] := 16#641B;
   // GBK_TO_UNICODE[32884] := 16#DEF7;
   // GBK_TO_UNICODE[32885] := 16#6420;
   // GBK_TO_UNICODE[32886] := 16#DEF8;
   // GBK_TO_UNICODE[32887] := 16#640C;
   // GBK_TO_UNICODE[32888] := 16#DEF9;
   // GBK_TO_UNICODE[32889] := 16#6426;
   // GBK_TO_UNICODE[32890] := 16#DEFA;
   // GBK_TO_UNICODE[32891] := 16#6421;
   // GBK_TO_UNICODE[32892] := 16#DEFB;
   // GBK_TO_UNICODE[32893] := 16#645E;
   // GBK_TO_UNICODE[32894] := 16#DEFC;
   // GBK_TO_UNICODE[32895] := 16#6484;
   // GBK_TO_UNICODE[32896] := 16#DEFD;
   // GBK_TO_UNICODE[32897] := 16#646D;
   // GBK_TO_UNICODE[32898] := 16#DEFE;
   // GBK_TO_UNICODE[32899] := 16#6496;
   // GBK_TO_UNICODE[32900] := 16#DF40;
   // GBK_TO_UNICODE[32901] := 16#9019;
   // GBK_TO_UNICODE[32902] := 16#DF41;
   // GBK_TO_UNICODE[32903] := 16#901C;
   // GBK_TO_UNICODE[32904] := 16#DF42;
   // GBK_TO_UNICODE[32905] := 16#9023;
   // GBK_TO_UNICODE[32906] := 16#DF43;
   // GBK_TO_UNICODE[32907] := 16#9024;
   // GBK_TO_UNICODE[32908] := 16#DF44;
   // GBK_TO_UNICODE[32909] := 16#9025;
   // GBK_TO_UNICODE[32910] := 16#DF45;
   // GBK_TO_UNICODE[32911] := 16#9027;
   // GBK_TO_UNICODE[32912] := 16#DF46;
   // GBK_TO_UNICODE[32913] := 16#9028;
   // GBK_TO_UNICODE[32914] := 16#DF47;
   // GBK_TO_UNICODE[32915] := 16#9029;
   // GBK_TO_UNICODE[32916] := 16#DF48;
   // GBK_TO_UNICODE[32917] := 16#902A;
   // GBK_TO_UNICODE[32918] := 16#DF49;
   // GBK_TO_UNICODE[32919] := 16#902B;
   // GBK_TO_UNICODE[32920] := 16#DF4A;
   // GBK_TO_UNICODE[32921] := 16#902C;
   // GBK_TO_UNICODE[32922] := 16#DF4B;
   // GBK_TO_UNICODE[32923] := 16#9030;
   // GBK_TO_UNICODE[32924] := 16#DF4C;
   // GBK_TO_UNICODE[32925] := 16#9031;
   // GBK_TO_UNICODE[32926] := 16#DF4D;
   // GBK_TO_UNICODE[32927] := 16#9032;
   // GBK_TO_UNICODE[32928] := 16#DF4E;
   // GBK_TO_UNICODE[32929] := 16#9033;
   // GBK_TO_UNICODE[32930] := 16#DF4F;
   // GBK_TO_UNICODE[32931] := 16#9034;
   // GBK_TO_UNICODE[32932] := 16#DF50;
   // GBK_TO_UNICODE[32933] := 16#9037;
   // GBK_TO_UNICODE[32934] := 16#DF51;
   // GBK_TO_UNICODE[32935] := 16#9039;
   // GBK_TO_UNICODE[32936] := 16#DF52;
   // GBK_TO_UNICODE[32937] := 16#903A;
   // GBK_TO_UNICODE[32938] := 16#DF53;
   // GBK_TO_UNICODE[32939] := 16#903D;
   // GBK_TO_UNICODE[32940] := 16#DF54;
   // GBK_TO_UNICODE[32941] := 16#903F;
   // GBK_TO_UNICODE[32942] := 16#DF55;
   // GBK_TO_UNICODE[32943] := 16#9040;
   // GBK_TO_UNICODE[32944] := 16#DF56;
   // GBK_TO_UNICODE[32945] := 16#9043;
   // GBK_TO_UNICODE[32946] := 16#DF57;
   // GBK_TO_UNICODE[32947] := 16#9045;
   // GBK_TO_UNICODE[32948] := 16#DF58;
   // GBK_TO_UNICODE[32949] := 16#9046;
   // GBK_TO_UNICODE[32950] := 16#DF59;
   // GBK_TO_UNICODE[32951] := 16#9048;
   // GBK_TO_UNICODE[32952] := 16#DF5A;
   // GBK_TO_UNICODE[32953] := 16#9049;
   // GBK_TO_UNICODE[32954] := 16#DF5B;
   // GBK_TO_UNICODE[32955] := 16#904A;
   // GBK_TO_UNICODE[32956] := 16#DF5C;
   // GBK_TO_UNICODE[32957] := 16#904B;
   // GBK_TO_UNICODE[32958] := 16#DF5D;
   // GBK_TO_UNICODE[32959] := 16#904C;
   // GBK_TO_UNICODE[32960] := 16#DF5E;
   // GBK_TO_UNICODE[32961] := 16#904E;
   // GBK_TO_UNICODE[32962] := 16#DF5F;
   // GBK_TO_UNICODE[32963] := 16#9054;
   // GBK_TO_UNICODE[32964] := 16#DF60;
   // GBK_TO_UNICODE[32965] := 16#9055;
   // GBK_TO_UNICODE[32966] := 16#DF61;
   // GBK_TO_UNICODE[32967] := 16#9056;
   // GBK_TO_UNICODE[32968] := 16#DF62;
   // GBK_TO_UNICODE[32969] := 16#9059;
   // GBK_TO_UNICODE[32970] := 16#DF63;
   // GBK_TO_UNICODE[32971] := 16#905A;
   // GBK_TO_UNICODE[32972] := 16#DF64;
   // GBK_TO_UNICODE[32973] := 16#905C;
   // GBK_TO_UNICODE[32974] := 16#DF65;
   // GBK_TO_UNICODE[32975] := 16#905D;
   // GBK_TO_UNICODE[32976] := 16#DF66;
   // GBK_TO_UNICODE[32977] := 16#905E;
   // GBK_TO_UNICODE[32978] := 16#DF67;
   // GBK_TO_UNICODE[32979] := 16#905F;
   // GBK_TO_UNICODE[32980] := 16#DF68;
   // GBK_TO_UNICODE[32981] := 16#9060;
   // GBK_TO_UNICODE[32982] := 16#DF69;
   // GBK_TO_UNICODE[32983] := 16#9061;
   // GBK_TO_UNICODE[32984] := 16#DF6A;
   // GBK_TO_UNICODE[32985] := 16#9064;
   // GBK_TO_UNICODE[32986] := 16#DF6B;
   // GBK_TO_UNICODE[32987] := 16#9066;
   // GBK_TO_UNICODE[32988] := 16#DF6C;
   // GBK_TO_UNICODE[32989] := 16#9067;
   // GBK_TO_UNICODE[32990] := 16#DF6D;
   // GBK_TO_UNICODE[32991] := 16#9069;
   // GBK_TO_UNICODE[32992] := 16#DF6E;
   // GBK_TO_UNICODE[32993] := 16#906A;
   // GBK_TO_UNICODE[32994] := 16#DF6F;
   // GBK_TO_UNICODE[32995] := 16#906B;
   // GBK_TO_UNICODE[32996] := 16#DF70;
   // GBK_TO_UNICODE[32997] := 16#906C;
   // GBK_TO_UNICODE[32998] := 16#DF71;
   // GBK_TO_UNICODE[32999] := 16#906F;
   // GBK_TO_UNICODE[33000] := 16#DF72;
   // GBK_TO_UNICODE[33001] := 16#9070;
   // GBK_TO_UNICODE[33002] := 16#DF73;
   // GBK_TO_UNICODE[33003] := 16#9071;
   // GBK_TO_UNICODE[33004] := 16#DF74;
   // GBK_TO_UNICODE[33005] := 16#9072;
   // GBK_TO_UNICODE[33006] := 16#DF75;
   // GBK_TO_UNICODE[33007] := 16#9073;
   // GBK_TO_UNICODE[33008] := 16#DF76;
   // GBK_TO_UNICODE[33009] := 16#9076;
   // GBK_TO_UNICODE[33010] := 16#DF77;
   // GBK_TO_UNICODE[33011] := 16#9077;
   // GBK_TO_UNICODE[33012] := 16#DF78;
   // GBK_TO_UNICODE[33013] := 16#9078;
   // GBK_TO_UNICODE[33014] := 16#DF79;
   // GBK_TO_UNICODE[33015] := 16#9079;
   // GBK_TO_UNICODE[33016] := 16#DF7A;
   // GBK_TO_UNICODE[33017] := 16#907A;
   // GBK_TO_UNICODE[33018] := 16#DF7B;
   // GBK_TO_UNICODE[33019] := 16#907B;
   // GBK_TO_UNICODE[33020] := 16#DF7C;
   // GBK_TO_UNICODE[33021] := 16#907C;
   // GBK_TO_UNICODE[33022] := 16#DF7D;
   // GBK_TO_UNICODE[33023] := 16#907E;
   // GBK_TO_UNICODE[33024] := 16#DF7E;
   // GBK_TO_UNICODE[33025] := 16#9081;
   // GBK_TO_UNICODE[33026] := 16#DF80;
   // GBK_TO_UNICODE[33027] := 16#9084;
   // GBK_TO_UNICODE[33028] := 16#DF81;
   // GBK_TO_UNICODE[33029] := 16#9085;
   // GBK_TO_UNICODE[33030] := 16#DF82;
   // GBK_TO_UNICODE[33031] := 16#9086;
   // GBK_TO_UNICODE[33032] := 16#DF83;
   // GBK_TO_UNICODE[33033] := 16#9087;
   // GBK_TO_UNICODE[33034] := 16#DF84;
   // GBK_TO_UNICODE[33035] := 16#9089;
   // GBK_TO_UNICODE[33036] := 16#DF85;
   // GBK_TO_UNICODE[33037] := 16#908A;
   // GBK_TO_UNICODE[33038] := 16#DF86;
   // GBK_TO_UNICODE[33039] := 16#908C;
   // GBK_TO_UNICODE[33040] := 16#DF87;
   // GBK_TO_UNICODE[33041] := 16#908D;
   // GBK_TO_UNICODE[33042] := 16#DF88;
   // GBK_TO_UNICODE[33043] := 16#908E;
   // GBK_TO_UNICODE[33044] := 16#DF89;
   // GBK_TO_UNICODE[33045] := 16#908F;
   // GBK_TO_UNICODE[33046] := 16#DF8A;
   // GBK_TO_UNICODE[33047] := 16#9090;
   // GBK_TO_UNICODE[33048] := 16#DF8B;
   // GBK_TO_UNICODE[33049] := 16#9092;
   // GBK_TO_UNICODE[33050] := 16#DF8C;
   // GBK_TO_UNICODE[33051] := 16#9094;
   // GBK_TO_UNICODE[33052] := 16#DF8D;
   // GBK_TO_UNICODE[33053] := 16#9096;
   // GBK_TO_UNICODE[33054] := 16#DF8E;
   // GBK_TO_UNICODE[33055] := 16#9098;
   // GBK_TO_UNICODE[33056] := 16#DF8F;
   // GBK_TO_UNICODE[33057] := 16#909A;
   // GBK_TO_UNICODE[33058] := 16#DF90;
   // GBK_TO_UNICODE[33059] := 16#909C;
   // GBK_TO_UNICODE[33060] := 16#DF91;
   // GBK_TO_UNICODE[33061] := 16#909E;
   // GBK_TO_UNICODE[33062] := 16#DF92;
   // GBK_TO_UNICODE[33063] := 16#909F;
   // GBK_TO_UNICODE[33064] := 16#DF93;
   // GBK_TO_UNICODE[33065] := 16#90A0;
   // GBK_TO_UNICODE[33066] := 16#DF94;
   // GBK_TO_UNICODE[33067] := 16#90A4;
   // GBK_TO_UNICODE[33068] := 16#DF95;
   // GBK_TO_UNICODE[33069] := 16#90A5;
   // GBK_TO_UNICODE[33070] := 16#DF96;
   // GBK_TO_UNICODE[33071] := 16#90A7;
   // GBK_TO_UNICODE[33072] := 16#DF97;
   // GBK_TO_UNICODE[33073] := 16#90A8;
   // GBK_TO_UNICODE[33074] := 16#DF98;
   // GBK_TO_UNICODE[33075] := 16#90A9;
   // GBK_TO_UNICODE[33076] := 16#DF99;
   // GBK_TO_UNICODE[33077] := 16#90AB;
   // GBK_TO_UNICODE[33078] := 16#DF9A;
   // GBK_TO_UNICODE[33079] := 16#90AD;
   // GBK_TO_UNICODE[33080] := 16#DF9B;
   // GBK_TO_UNICODE[33081] := 16#90B2;
   // GBK_TO_UNICODE[33082] := 16#DF9C;
   // GBK_TO_UNICODE[33083] := 16#90B7;
   // GBK_TO_UNICODE[33084] := 16#DF9D;
   // GBK_TO_UNICODE[33085] := 16#90BC;
   // GBK_TO_UNICODE[33086] := 16#DF9E;
   // GBK_TO_UNICODE[33087] := 16#90BD;
   // GBK_TO_UNICODE[33088] := 16#DF9F;
   // GBK_TO_UNICODE[33089] := 16#90BF;
   // GBK_TO_UNICODE[33090] := 16#DFA0;
   // GBK_TO_UNICODE[33091] := 16#90C0;
   // GBK_TO_UNICODE[33092] := 16#DFA1;
   // GBK_TO_UNICODE[33093] := 16#647A;
   // GBK_TO_UNICODE[33094] := 16#DFA2;
   // GBK_TO_UNICODE[33095] := 16#64B7;
   // GBK_TO_UNICODE[33096] := 16#DFA3;
   // GBK_TO_UNICODE[33097] := 16#64B8;
   // GBK_TO_UNICODE[33098] := 16#DFA4;
   // GBK_TO_UNICODE[33099] := 16#6499;
   // GBK_TO_UNICODE[33100] := 16#DFA5;
   // GBK_TO_UNICODE[33101] := 16#64BA;
   // GBK_TO_UNICODE[33102] := 16#DFA6;
   // GBK_TO_UNICODE[33103] := 16#64C0;
   // GBK_TO_UNICODE[33104] := 16#DFA7;
   // GBK_TO_UNICODE[33105] := 16#64D0;
   // GBK_TO_UNICODE[33106] := 16#DFA8;
   // GBK_TO_UNICODE[33107] := 16#64D7;
   // GBK_TO_UNICODE[33108] := 16#DFA9;
   // GBK_TO_UNICODE[33109] := 16#64E4;
   // GBK_TO_UNICODE[33110] := 16#DFAA;
   // GBK_TO_UNICODE[33111] := 16#64E2;
   // GBK_TO_UNICODE[33112] := 16#DFAB;
   // GBK_TO_UNICODE[33113] := 16#6509;
   // GBK_TO_UNICODE[33114] := 16#DFAC;
   // GBK_TO_UNICODE[33115] := 16#6525;
   // GBK_TO_UNICODE[33116] := 16#DFAD;
   // GBK_TO_UNICODE[33117] := 16#652E;
   // GBK_TO_UNICODE[33118] := 16#DFAE;
   // GBK_TO_UNICODE[33119] := 16#5F0B;
   // GBK_TO_UNICODE[33120] := 16#DFAF;
   // GBK_TO_UNICODE[33121] := 16#5FD2;
   // GBK_TO_UNICODE[33122] := 16#DFB0;
   // GBK_TO_UNICODE[33123] := 16#7519;
   // GBK_TO_UNICODE[33124] := 16#DFB1;
   // GBK_TO_UNICODE[33125] := 16#5F11;
   // GBK_TO_UNICODE[33126] := 16#DFB2;
   // GBK_TO_UNICODE[33127] := 16#535F;
   // GBK_TO_UNICODE[33128] := 16#DFB3;
   // GBK_TO_UNICODE[33129] := 16#53F1;
   // GBK_TO_UNICODE[33130] := 16#DFB4;
   // GBK_TO_UNICODE[33131] := 16#53FD;
   // GBK_TO_UNICODE[33132] := 16#DFB5;
   // GBK_TO_UNICODE[33133] := 16#53E9;
   // GBK_TO_UNICODE[33134] := 16#DFB6;
   // GBK_TO_UNICODE[33135] := 16#53E8;
   // GBK_TO_UNICODE[33136] := 16#DFB7;
   // GBK_TO_UNICODE[33137] := 16#53FB;
   // GBK_TO_UNICODE[33138] := 16#DFB8;
   // GBK_TO_UNICODE[33139] := 16#5412;
   // GBK_TO_UNICODE[33140] := 16#DFB9;
   // GBK_TO_UNICODE[33141] := 16#5416;
   // GBK_TO_UNICODE[33142] := 16#DFBA;
   // GBK_TO_UNICODE[33143] := 16#5406;
   // GBK_TO_UNICODE[33144] := 16#DFBB;
   // GBK_TO_UNICODE[33145] := 16#544B;
   // GBK_TO_UNICODE[33146] := 16#DFBC;
   // GBK_TO_UNICODE[33147] := 16#5452;
   // GBK_TO_UNICODE[33148] := 16#DFBD;
   // GBK_TO_UNICODE[33149] := 16#5453;
   // GBK_TO_UNICODE[33150] := 16#DFBE;
   // GBK_TO_UNICODE[33151] := 16#5454;
   // GBK_TO_UNICODE[33152] := 16#DFBF;
   // GBK_TO_UNICODE[33153] := 16#5456;
   // GBK_TO_UNICODE[33154] := 16#DFC0;
   // GBK_TO_UNICODE[33155] := 16#5443;
   // GBK_TO_UNICODE[33156] := 16#DFC1;
   // GBK_TO_UNICODE[33157] := 16#5421;
   // GBK_TO_UNICODE[33158] := 16#DFC2;
   // GBK_TO_UNICODE[33159] := 16#5457;
   // GBK_TO_UNICODE[33160] := 16#DFC3;
   // GBK_TO_UNICODE[33161] := 16#5459;
   // GBK_TO_UNICODE[33162] := 16#DFC4;
   // GBK_TO_UNICODE[33163] := 16#5423;
   // GBK_TO_UNICODE[33164] := 16#DFC5;
   // GBK_TO_UNICODE[33165] := 16#5432;
   // GBK_TO_UNICODE[33166] := 16#DFC6;
   // GBK_TO_UNICODE[33167] := 16#5482;
   // GBK_TO_UNICODE[33168] := 16#DFC7;
   // GBK_TO_UNICODE[33169] := 16#5494;
   // GBK_TO_UNICODE[33170] := 16#DFC8;
   // GBK_TO_UNICODE[33171] := 16#5477;
   // GBK_TO_UNICODE[33172] := 16#DFC9;
   // GBK_TO_UNICODE[33173] := 16#5471;
   // GBK_TO_UNICODE[33174] := 16#DFCA;
   // GBK_TO_UNICODE[33175] := 16#5464;
   // GBK_TO_UNICODE[33176] := 16#DFCB;
   // GBK_TO_UNICODE[33177] := 16#549A;
   // GBK_TO_UNICODE[33178] := 16#DFCC;
   // GBK_TO_UNICODE[33179] := 16#549B;
   // GBK_TO_UNICODE[33180] := 16#DFCD;
   // GBK_TO_UNICODE[33181] := 16#5484;
   // GBK_TO_UNICODE[33182] := 16#DFCE;
   // GBK_TO_UNICODE[33183] := 16#5476;
   // GBK_TO_UNICODE[33184] := 16#DFCF;
   // GBK_TO_UNICODE[33185] := 16#5466;
   // GBK_TO_UNICODE[33186] := 16#DFD0;
   // GBK_TO_UNICODE[33187] := 16#549D;
   // GBK_TO_UNICODE[33188] := 16#DFD1;
   // GBK_TO_UNICODE[33189] := 16#54D0;
   // GBK_TO_UNICODE[33190] := 16#DFD2;
   // GBK_TO_UNICODE[33191] := 16#54AD;
   // GBK_TO_UNICODE[33192] := 16#DFD3;
   // GBK_TO_UNICODE[33193] := 16#54C2;
   // GBK_TO_UNICODE[33194] := 16#DFD4;
   // GBK_TO_UNICODE[33195] := 16#54B4;
   // GBK_TO_UNICODE[33196] := 16#DFD5;
   // GBK_TO_UNICODE[33197] := 16#54D2;
   // GBK_TO_UNICODE[33198] := 16#DFD6;
   // GBK_TO_UNICODE[33199] := 16#54A7;
   // GBK_TO_UNICODE[33200] := 16#DFD7;
   // GBK_TO_UNICODE[33201] := 16#54A6;
   // GBK_TO_UNICODE[33202] := 16#DFD8;
   // GBK_TO_UNICODE[33203] := 16#54D3;
   // GBK_TO_UNICODE[33204] := 16#DFD9;
   // GBK_TO_UNICODE[33205] := 16#54D4;
   // GBK_TO_UNICODE[33206] := 16#DFDA;
   // GBK_TO_UNICODE[33207] := 16#5472;
   // GBK_TO_UNICODE[33208] := 16#DFDB;
   // GBK_TO_UNICODE[33209] := 16#54A3;
   // GBK_TO_UNICODE[33210] := 16#DFDC;
   // GBK_TO_UNICODE[33211] := 16#54D5;
   // GBK_TO_UNICODE[33212] := 16#DFDD;
   // GBK_TO_UNICODE[33213] := 16#54BB;
   // GBK_TO_UNICODE[33214] := 16#DFDE;
   // GBK_TO_UNICODE[33215] := 16#54BF;
   // GBK_TO_UNICODE[33216] := 16#DFDF;
   // GBK_TO_UNICODE[33217] := 16#54CC;
   // GBK_TO_UNICODE[33218] := 16#DFE0;
   // GBK_TO_UNICODE[33219] := 16#54D9;
   // GBK_TO_UNICODE[33220] := 16#DFE1;
   // GBK_TO_UNICODE[33221] := 16#54DA;
   // GBK_TO_UNICODE[33222] := 16#DFE2;
   // GBK_TO_UNICODE[33223] := 16#54DC;
   // GBK_TO_UNICODE[33224] := 16#DFE3;
   // GBK_TO_UNICODE[33225] := 16#54A9;
   // GBK_TO_UNICODE[33226] := 16#DFE4;
   // GBK_TO_UNICODE[33227] := 16#54AA;
   // GBK_TO_UNICODE[33228] := 16#DFE5;
   // GBK_TO_UNICODE[33229] := 16#54A4;
   // GBK_TO_UNICODE[33230] := 16#DFE6;
   // GBK_TO_UNICODE[33231] := 16#54DD;
   // GBK_TO_UNICODE[33232] := 16#DFE7;
   // GBK_TO_UNICODE[33233] := 16#54CF;
   // GBK_TO_UNICODE[33234] := 16#DFE8;
   // GBK_TO_UNICODE[33235] := 16#54DE;
   // GBK_TO_UNICODE[33236] := 16#DFE9;
   // GBK_TO_UNICODE[33237] := 16#551B;
   // GBK_TO_UNICODE[33238] := 16#DFEA;
   // GBK_TO_UNICODE[33239] := 16#54E7;
   // GBK_TO_UNICODE[33240] := 16#DFEB;
   // GBK_TO_UNICODE[33241] := 16#5520;
   // GBK_TO_UNICODE[33242] := 16#DFEC;
   // GBK_TO_UNICODE[33243] := 16#54FD;
   // GBK_TO_UNICODE[33244] := 16#DFED;
   // GBK_TO_UNICODE[33245] := 16#5514;
   // GBK_TO_UNICODE[33246] := 16#DFEE;
   // GBK_TO_UNICODE[33247] := 16#54F3;
   // GBK_TO_UNICODE[33248] := 16#DFEF;
   // GBK_TO_UNICODE[33249] := 16#5522;
   // GBK_TO_UNICODE[33250] := 16#DFF0;
   // GBK_TO_UNICODE[33251] := 16#5523;
   // GBK_TO_UNICODE[33252] := 16#DFF1;
   // GBK_TO_UNICODE[33253] := 16#550F;
   // GBK_TO_UNICODE[33254] := 16#DFF2;
   // GBK_TO_UNICODE[33255] := 16#5511;
   // GBK_TO_UNICODE[33256] := 16#DFF3;
   // GBK_TO_UNICODE[33257] := 16#5527;
   // GBK_TO_UNICODE[33258] := 16#DFF4;
   // GBK_TO_UNICODE[33259] := 16#552A;
   // GBK_TO_UNICODE[33260] := 16#DFF5;
   // GBK_TO_UNICODE[33261] := 16#5567;
   // GBK_TO_UNICODE[33262] := 16#DFF6;
   // GBK_TO_UNICODE[33263] := 16#558F;
   // GBK_TO_UNICODE[33264] := 16#DFF7;
   // GBK_TO_UNICODE[33265] := 16#55B5;
   // GBK_TO_UNICODE[33266] := 16#DFF8;
   // GBK_TO_UNICODE[33267] := 16#5549;
   // GBK_TO_UNICODE[33268] := 16#DFF9;
   // GBK_TO_UNICODE[33269] := 16#556D;
   // GBK_TO_UNICODE[33270] := 16#DFFA;
   // GBK_TO_UNICODE[33271] := 16#5541;
   // GBK_TO_UNICODE[33272] := 16#DFFB;
   // GBK_TO_UNICODE[33273] := 16#5555;
   // GBK_TO_UNICODE[33274] := 16#DFFC;
   // GBK_TO_UNICODE[33275] := 16#553F;
   // GBK_TO_UNICODE[33276] := 16#DFFD;
   // GBK_TO_UNICODE[33277] := 16#5550;
   // GBK_TO_UNICODE[33278] := 16#DFFE;
   // GBK_TO_UNICODE[33279] := 16#553C;
   // GBK_TO_UNICODE[33280] := 16#E040;
   // GBK_TO_UNICODE[33281] := 16#90C2;
   // GBK_TO_UNICODE[33282] := 16#E041;
   // GBK_TO_UNICODE[33283] := 16#90C3;
   // GBK_TO_UNICODE[33284] := 16#E042;
   // GBK_TO_UNICODE[33285] := 16#90C6;
   // GBK_TO_UNICODE[33286] := 16#E043;
   // GBK_TO_UNICODE[33287] := 16#90C8;
   // GBK_TO_UNICODE[33288] := 16#E044;
   // GBK_TO_UNICODE[33289] := 16#90C9;
   // GBK_TO_UNICODE[33290] := 16#E045;
   // GBK_TO_UNICODE[33291] := 16#90CB;
   // GBK_TO_UNICODE[33292] := 16#E046;
   // GBK_TO_UNICODE[33293] := 16#90CC;
   // GBK_TO_UNICODE[33294] := 16#E047;
   // GBK_TO_UNICODE[33295] := 16#90CD;
   // GBK_TO_UNICODE[33296] := 16#E048;
   // GBK_TO_UNICODE[33297] := 16#90D2;
   // GBK_TO_UNICODE[33298] := 16#E049;
   // GBK_TO_UNICODE[33299] := 16#90D4;
   // GBK_TO_UNICODE[33300] := 16#E04A;
   // GBK_TO_UNICODE[33301] := 16#90D5;
   // GBK_TO_UNICODE[33302] := 16#E04B;
   // GBK_TO_UNICODE[33303] := 16#90D6;
   // GBK_TO_UNICODE[33304] := 16#E04C;
   // GBK_TO_UNICODE[33305] := 16#90D8;
   // GBK_TO_UNICODE[33306] := 16#E04D;
   // GBK_TO_UNICODE[33307] := 16#90D9;
   // GBK_TO_UNICODE[33308] := 16#E04E;
   // GBK_TO_UNICODE[33309] := 16#90DA;
   // GBK_TO_UNICODE[33310] := 16#E04F;
   // GBK_TO_UNICODE[33311] := 16#90DE;
   // GBK_TO_UNICODE[33312] := 16#E050;
   // GBK_TO_UNICODE[33313] := 16#90DF;
   // GBK_TO_UNICODE[33314] := 16#E051;
   // GBK_TO_UNICODE[33315] := 16#90E0;
   // GBK_TO_UNICODE[33316] := 16#E052;
   // GBK_TO_UNICODE[33317] := 16#90E3;
   // GBK_TO_UNICODE[33318] := 16#E053;
   // GBK_TO_UNICODE[33319] := 16#90E4;
   // GBK_TO_UNICODE[33320] := 16#E054;
   // GBK_TO_UNICODE[33321] := 16#90E5;
   // GBK_TO_UNICODE[33322] := 16#E055;
   // GBK_TO_UNICODE[33323] := 16#90E9;
   // GBK_TO_UNICODE[33324] := 16#E056;
   // GBK_TO_UNICODE[33325] := 16#90EA;
   // GBK_TO_UNICODE[33326] := 16#E057;
   // GBK_TO_UNICODE[33327] := 16#90EC;
   // GBK_TO_UNICODE[33328] := 16#E058;
   // GBK_TO_UNICODE[33329] := 16#90EE;
   // GBK_TO_UNICODE[33330] := 16#E059;
   // GBK_TO_UNICODE[33331] := 16#90F0;
   // GBK_TO_UNICODE[33332] := 16#E05A;
   // GBK_TO_UNICODE[33333] := 16#90F1;
   // GBK_TO_UNICODE[33334] := 16#E05B;
   // GBK_TO_UNICODE[33335] := 16#90F2;
   // GBK_TO_UNICODE[33336] := 16#E05C;
   // GBK_TO_UNICODE[33337] := 16#90F3;
   // GBK_TO_UNICODE[33338] := 16#E05D;
   // GBK_TO_UNICODE[33339] := 16#90F5;
   // GBK_TO_UNICODE[33340] := 16#E05E;
   // GBK_TO_UNICODE[33341] := 16#90F6;
   // GBK_TO_UNICODE[33342] := 16#E05F;
   // GBK_TO_UNICODE[33343] := 16#90F7;
   // GBK_TO_UNICODE[33344] := 16#E060;
   // GBK_TO_UNICODE[33345] := 16#90F9;
   // GBK_TO_UNICODE[33346] := 16#E061;
   // GBK_TO_UNICODE[33347] := 16#90FA;
   // GBK_TO_UNICODE[33348] := 16#E062;
   // GBK_TO_UNICODE[33349] := 16#90FB;
   // GBK_TO_UNICODE[33350] := 16#E063;
   // GBK_TO_UNICODE[33351] := 16#90FC;
   // GBK_TO_UNICODE[33352] := 16#E064;
   // GBK_TO_UNICODE[33353] := 16#90FF;
   // GBK_TO_UNICODE[33354] := 16#E065;
   // GBK_TO_UNICODE[33355] := 16#9100;
   // GBK_TO_UNICODE[33356] := 16#E066;
   // GBK_TO_UNICODE[33357] := 16#9101;
   // GBK_TO_UNICODE[33358] := 16#E067;
   // GBK_TO_UNICODE[33359] := 16#9103;
   // GBK_TO_UNICODE[33360] := 16#E068;
   // GBK_TO_UNICODE[33361] := 16#9105;
   // GBK_TO_UNICODE[33362] := 16#E069;
   // GBK_TO_UNICODE[33363] := 16#9106;
   // GBK_TO_UNICODE[33364] := 16#E06A;
   // GBK_TO_UNICODE[33365] := 16#9107;
   // GBK_TO_UNICODE[33366] := 16#E06B;
   // GBK_TO_UNICODE[33367] := 16#9108;
   // GBK_TO_UNICODE[33368] := 16#E06C;
   // GBK_TO_UNICODE[33369] := 16#9109;
   // GBK_TO_UNICODE[33370] := 16#E06D;
   // GBK_TO_UNICODE[33371] := 16#910A;
   // GBK_TO_UNICODE[33372] := 16#E06E;
   // GBK_TO_UNICODE[33373] := 16#910B;
   // GBK_TO_UNICODE[33374] := 16#E06F;
   // GBK_TO_UNICODE[33375] := 16#910C;
   // GBK_TO_UNICODE[33376] := 16#E070;
   // GBK_TO_UNICODE[33377] := 16#910D;
   // GBK_TO_UNICODE[33378] := 16#E071;
   // GBK_TO_UNICODE[33379] := 16#910E;
   // GBK_TO_UNICODE[33380] := 16#E072;
   // GBK_TO_UNICODE[33381] := 16#910F;
   // GBK_TO_UNICODE[33382] := 16#E073;
   // GBK_TO_UNICODE[33383] := 16#9110;
   // GBK_TO_UNICODE[33384] := 16#E074;
   // GBK_TO_UNICODE[33385] := 16#9111;
   // GBK_TO_UNICODE[33386] := 16#E075;
   // GBK_TO_UNICODE[33387] := 16#9112;
   // GBK_TO_UNICODE[33388] := 16#E076;
   // GBK_TO_UNICODE[33389] := 16#9113;
   // GBK_TO_UNICODE[33390] := 16#E077;
   // GBK_TO_UNICODE[33391] := 16#9114;
   // GBK_TO_UNICODE[33392] := 16#E078;
   // GBK_TO_UNICODE[33393] := 16#9115;
   // GBK_TO_UNICODE[33394] := 16#E079;
   // GBK_TO_UNICODE[33395] := 16#9116;
   // GBK_TO_UNICODE[33396] := 16#E07A;
   // GBK_TO_UNICODE[33397] := 16#9117;
   // GBK_TO_UNICODE[33398] := 16#E07B;
   // GBK_TO_UNICODE[33399] := 16#9118;
   // GBK_TO_UNICODE[33400] := 16#E07C;
   // GBK_TO_UNICODE[33401] := 16#911A;
   // GBK_TO_UNICODE[33402] := 16#E07D;
   // GBK_TO_UNICODE[33403] := 16#911B;
   // GBK_TO_UNICODE[33404] := 16#E07E;
   // GBK_TO_UNICODE[33405] := 16#911C;
   // GBK_TO_UNICODE[33406] := 16#E080;
   // GBK_TO_UNICODE[33407] := 16#911D;
   // GBK_TO_UNICODE[33408] := 16#E081;
   // GBK_TO_UNICODE[33409] := 16#911F;
   // GBK_TO_UNICODE[33410] := 16#E082;
   // GBK_TO_UNICODE[33411] := 16#9120;
   // GBK_TO_UNICODE[33412] := 16#E083;
   // GBK_TO_UNICODE[33413] := 16#9121;
   // GBK_TO_UNICODE[33414] := 16#E084;
   // GBK_TO_UNICODE[33415] := 16#9124;
   // GBK_TO_UNICODE[33416] := 16#E085;
   // GBK_TO_UNICODE[33417] := 16#9125;
   // GBK_TO_UNICODE[33418] := 16#E086;
   // GBK_TO_UNICODE[33419] := 16#9126;
   // GBK_TO_UNICODE[33420] := 16#E087;
   // GBK_TO_UNICODE[33421] := 16#9127;
   // GBK_TO_UNICODE[33422] := 16#E088;
   // GBK_TO_UNICODE[33423] := 16#9128;
   // GBK_TO_UNICODE[33424] := 16#E089;
   // GBK_TO_UNICODE[33425] := 16#9129;
   // GBK_TO_UNICODE[33426] := 16#E08A;
   // GBK_TO_UNICODE[33427] := 16#912A;
   // GBK_TO_UNICODE[33428] := 16#E08B;
   // GBK_TO_UNICODE[33429] := 16#912B;
   // GBK_TO_UNICODE[33430] := 16#E08C;
   // GBK_TO_UNICODE[33431] := 16#912C;
   // GBK_TO_UNICODE[33432] := 16#E08D;
   // GBK_TO_UNICODE[33433] := 16#912D;
   // GBK_TO_UNICODE[33434] := 16#E08E;
   // GBK_TO_UNICODE[33435] := 16#912E;
   // GBK_TO_UNICODE[33436] := 16#E08F;
   // GBK_TO_UNICODE[33437] := 16#9130;
   // GBK_TO_UNICODE[33438] := 16#E090;
   // GBK_TO_UNICODE[33439] := 16#9132;
   // GBK_TO_UNICODE[33440] := 16#E091;
   // GBK_TO_UNICODE[33441] := 16#9133;
   // GBK_TO_UNICODE[33442] := 16#E092;
   // GBK_TO_UNICODE[33443] := 16#9134;
   // GBK_TO_UNICODE[33444] := 16#E093;
   // GBK_TO_UNICODE[33445] := 16#9135;
   // GBK_TO_UNICODE[33446] := 16#E094;
   // GBK_TO_UNICODE[33447] := 16#9136;
   // GBK_TO_UNICODE[33448] := 16#E095;
   // GBK_TO_UNICODE[33449] := 16#9137;
   // GBK_TO_UNICODE[33450] := 16#E096;
   // GBK_TO_UNICODE[33451] := 16#9138;
   // GBK_TO_UNICODE[33452] := 16#E097;
   // GBK_TO_UNICODE[33453] := 16#913A;
   // GBK_TO_UNICODE[33454] := 16#E098;
   // GBK_TO_UNICODE[33455] := 16#913B;
   // GBK_TO_UNICODE[33456] := 16#E099;
   // GBK_TO_UNICODE[33457] := 16#913C;
   // GBK_TO_UNICODE[33458] := 16#E09A;
   // GBK_TO_UNICODE[33459] := 16#913D;
   // GBK_TO_UNICODE[33460] := 16#E09B;
   // GBK_TO_UNICODE[33461] := 16#913E;
   // GBK_TO_UNICODE[33462] := 16#E09C;
   // GBK_TO_UNICODE[33463] := 16#913F;
   // GBK_TO_UNICODE[33464] := 16#E09D;
   // GBK_TO_UNICODE[33465] := 16#9140;
   // GBK_TO_UNICODE[33466] := 16#E09E;
   // GBK_TO_UNICODE[33467] := 16#9141;
   // GBK_TO_UNICODE[33468] := 16#E09F;
   // GBK_TO_UNICODE[33469] := 16#9142;
   // GBK_TO_UNICODE[33470] := 16#E0A0;
   // GBK_TO_UNICODE[33471] := 16#9144;
   // GBK_TO_UNICODE[33472] := 16#E0A1;
   // GBK_TO_UNICODE[33473] := 16#5537;
   // GBK_TO_UNICODE[33474] := 16#E0A2;
   // GBK_TO_UNICODE[33475] := 16#5556;
   // GBK_TO_UNICODE[33476] := 16#E0A3;
   // GBK_TO_UNICODE[33477] := 16#5575;
   // GBK_TO_UNICODE[33478] := 16#E0A4;
   // GBK_TO_UNICODE[33479] := 16#5576;
   // GBK_TO_UNICODE[33480] := 16#E0A5;
   // GBK_TO_UNICODE[33481] := 16#5577;
   // GBK_TO_UNICODE[33482] := 16#E0A6;
   // GBK_TO_UNICODE[33483] := 16#5533;
   // GBK_TO_UNICODE[33484] := 16#E0A7;
   // GBK_TO_UNICODE[33485] := 16#5530;
   // GBK_TO_UNICODE[33486] := 16#E0A8;
   // GBK_TO_UNICODE[33487] := 16#555C;
   // GBK_TO_UNICODE[33488] := 16#E0A9;
   // GBK_TO_UNICODE[33489] := 16#558B;
   // GBK_TO_UNICODE[33490] := 16#E0AA;
   // GBK_TO_UNICODE[33491] := 16#55D2;
   // GBK_TO_UNICODE[33492] := 16#E0AB;
   // GBK_TO_UNICODE[33493] := 16#5583;
   // GBK_TO_UNICODE[33494] := 16#E0AC;
   // GBK_TO_UNICODE[33495] := 16#55B1;
   // GBK_TO_UNICODE[33496] := 16#E0AD;
   // GBK_TO_UNICODE[33497] := 16#55B9;
   // GBK_TO_UNICODE[33498] := 16#E0AE;
   // GBK_TO_UNICODE[33499] := 16#5588;
   // GBK_TO_UNICODE[33500] := 16#E0AF;
   // GBK_TO_UNICODE[33501] := 16#5581;
   // GBK_TO_UNICODE[33502] := 16#E0B0;
   // GBK_TO_UNICODE[33503] := 16#559F;
   // GBK_TO_UNICODE[33504] := 16#E0B1;
   // GBK_TO_UNICODE[33505] := 16#557E;
   // GBK_TO_UNICODE[33506] := 16#E0B2;
   // GBK_TO_UNICODE[33507] := 16#55D6;
   // GBK_TO_UNICODE[33508] := 16#E0B3;
   // GBK_TO_UNICODE[33509] := 16#5591;
   // GBK_TO_UNICODE[33510] := 16#E0B4;
   // GBK_TO_UNICODE[33511] := 16#557B;
   // GBK_TO_UNICODE[33512] := 16#E0B5;
   // GBK_TO_UNICODE[33513] := 16#55DF;
   // GBK_TO_UNICODE[33514] := 16#E0B6;
   // GBK_TO_UNICODE[33515] := 16#55BD;
   // GBK_TO_UNICODE[33516] := 16#E0B7;
   // GBK_TO_UNICODE[33517] := 16#55BE;
   // GBK_TO_UNICODE[33518] := 16#E0B8;
   // GBK_TO_UNICODE[33519] := 16#5594;
   // GBK_TO_UNICODE[33520] := 16#E0B9;
   // GBK_TO_UNICODE[33521] := 16#5599;
   // GBK_TO_UNICODE[33522] := 16#E0BA;
   // GBK_TO_UNICODE[33523] := 16#55EA;
   // GBK_TO_UNICODE[33524] := 16#E0BB;
   // GBK_TO_UNICODE[33525] := 16#55F7;
   // GBK_TO_UNICODE[33526] := 16#E0BC;
   // GBK_TO_UNICODE[33527] := 16#55C9;
   // GBK_TO_UNICODE[33528] := 16#E0BD;
   // GBK_TO_UNICODE[33529] := 16#561F;
   // GBK_TO_UNICODE[33530] := 16#E0BE;
   // GBK_TO_UNICODE[33531] := 16#55D1;
   // GBK_TO_UNICODE[33532] := 16#E0BF;
   // GBK_TO_UNICODE[33533] := 16#55EB;
   // GBK_TO_UNICODE[33534] := 16#E0C0;
   // GBK_TO_UNICODE[33535] := 16#55EC;
   // GBK_TO_UNICODE[33536] := 16#E0C1;
   // GBK_TO_UNICODE[33537] := 16#55D4;
   // GBK_TO_UNICODE[33538] := 16#E0C2;
   // GBK_TO_UNICODE[33539] := 16#55E6;
   // GBK_TO_UNICODE[33540] := 16#E0C3;
   // GBK_TO_UNICODE[33541] := 16#55DD;
   // GBK_TO_UNICODE[33542] := 16#E0C4;
   // GBK_TO_UNICODE[33543] := 16#55C4;
   // GBK_TO_UNICODE[33544] := 16#E0C5;
   // GBK_TO_UNICODE[33545] := 16#55EF;
   // GBK_TO_UNICODE[33546] := 16#E0C6;
   // GBK_TO_UNICODE[33547] := 16#55E5;
   // GBK_TO_UNICODE[33548] := 16#E0C7;
   // GBK_TO_UNICODE[33549] := 16#55F2;
   // GBK_TO_UNICODE[33550] := 16#E0C8;
   // GBK_TO_UNICODE[33551] := 16#55F3;
   // GBK_TO_UNICODE[33552] := 16#E0C9;
   // GBK_TO_UNICODE[33553] := 16#55CC;
   // GBK_TO_UNICODE[33554] := 16#E0CA;
   // GBK_TO_UNICODE[33555] := 16#55CD;
   // GBK_TO_UNICODE[33556] := 16#E0CB;
   // GBK_TO_UNICODE[33557] := 16#55E8;
   // GBK_TO_UNICODE[33558] := 16#E0CC;
   // GBK_TO_UNICODE[33559] := 16#55F5;
   // GBK_TO_UNICODE[33560] := 16#E0CD;
   // GBK_TO_UNICODE[33561] := 16#55E4;
   // GBK_TO_UNICODE[33562] := 16#E0CE;
   // GBK_TO_UNICODE[33563] := 16#8F94;
   // GBK_TO_UNICODE[33564] := 16#E0CF;
   // GBK_TO_UNICODE[33565] := 16#561E;
   // GBK_TO_UNICODE[33566] := 16#E0D0;
   // GBK_TO_UNICODE[33567] := 16#5608;
   // GBK_TO_UNICODE[33568] := 16#E0D1;
   // GBK_TO_UNICODE[33569] := 16#560C;
   // GBK_TO_UNICODE[33570] := 16#E0D2;
   // GBK_TO_UNICODE[33571] := 16#5601;
   // GBK_TO_UNICODE[33572] := 16#E0D3;
   // GBK_TO_UNICODE[33573] := 16#5624;
   // GBK_TO_UNICODE[33574] := 16#E0D4;
   // GBK_TO_UNICODE[33575] := 16#5623;
   // GBK_TO_UNICODE[33576] := 16#E0D5;
   // GBK_TO_UNICODE[33577] := 16#55FE;
   // GBK_TO_UNICODE[33578] := 16#E0D6;
   // GBK_TO_UNICODE[33579] := 16#5600;
   // GBK_TO_UNICODE[33580] := 16#E0D7;
   // GBK_TO_UNICODE[33581] := 16#5627;
   // GBK_TO_UNICODE[33582] := 16#E0D8;
   // GBK_TO_UNICODE[33583] := 16#562D;
   // GBK_TO_UNICODE[33584] := 16#E0D9;
   // GBK_TO_UNICODE[33585] := 16#5658;
   // GBK_TO_UNICODE[33586] := 16#E0DA;
   // GBK_TO_UNICODE[33587] := 16#5639;
   // GBK_TO_UNICODE[33588] := 16#E0DB;
   // GBK_TO_UNICODE[33589] := 16#5657;
   // GBK_TO_UNICODE[33590] := 16#E0DC;
   // GBK_TO_UNICODE[33591] := 16#562C;
   // GBK_TO_UNICODE[33592] := 16#E0DD;
   // GBK_TO_UNICODE[33593] := 16#564D;
   // GBK_TO_UNICODE[33594] := 16#E0DE;
   // GBK_TO_UNICODE[33595] := 16#5662;
   // GBK_TO_UNICODE[33596] := 16#E0DF;
   // GBK_TO_UNICODE[33597] := 16#5659;
   // GBK_TO_UNICODE[33598] := 16#E0E0;
   // GBK_TO_UNICODE[33599] := 16#565C;
   // GBK_TO_UNICODE[33600] := 16#E0E1;
   // GBK_TO_UNICODE[33601] := 16#564C;
   // GBK_TO_UNICODE[33602] := 16#E0E2;
   // GBK_TO_UNICODE[33603] := 16#5654;
   // GBK_TO_UNICODE[33604] := 16#E0E3;
   // GBK_TO_UNICODE[33605] := 16#5686;
   // GBK_TO_UNICODE[33606] := 16#E0E4;
   // GBK_TO_UNICODE[33607] := 16#5664;
   // GBK_TO_UNICODE[33608] := 16#E0E5;
   // GBK_TO_UNICODE[33609] := 16#5671;
   // GBK_TO_UNICODE[33610] := 16#E0E6;
   // GBK_TO_UNICODE[33611] := 16#566B;
   // GBK_TO_UNICODE[33612] := 16#E0E7;
   // GBK_TO_UNICODE[33613] := 16#567B;
   // GBK_TO_UNICODE[33614] := 16#E0E8;
   // GBK_TO_UNICODE[33615] := 16#567C;
   // GBK_TO_UNICODE[33616] := 16#E0E9;
   // GBK_TO_UNICODE[33617] := 16#5685;
   // GBK_TO_UNICODE[33618] := 16#E0EA;
   // GBK_TO_UNICODE[33619] := 16#5693;
   // GBK_TO_UNICODE[33620] := 16#E0EB;
   // GBK_TO_UNICODE[33621] := 16#56AF;
   // GBK_TO_UNICODE[33622] := 16#E0EC;
   // GBK_TO_UNICODE[33623] := 16#56D4;
   // GBK_TO_UNICODE[33624] := 16#E0ED;
   // GBK_TO_UNICODE[33625] := 16#56D7;
   // GBK_TO_UNICODE[33626] := 16#E0EE;
   // GBK_TO_UNICODE[33627] := 16#56DD;
   // GBK_TO_UNICODE[33628] := 16#E0EF;
   // GBK_TO_UNICODE[33629] := 16#56E1;
   // GBK_TO_UNICODE[33630] := 16#E0F0;
   // GBK_TO_UNICODE[33631] := 16#56F5;
   // GBK_TO_UNICODE[33632] := 16#E0F1;
   // GBK_TO_UNICODE[33633] := 16#56EB;
   // GBK_TO_UNICODE[33634] := 16#E0F2;
   // GBK_TO_UNICODE[33635] := 16#56F9;
   // GBK_TO_UNICODE[33636] := 16#E0F3;
   // GBK_TO_UNICODE[33637] := 16#56FF;
   // GBK_TO_UNICODE[33638] := 16#E0F4;
   // GBK_TO_UNICODE[33639] := 16#5704;
   // GBK_TO_UNICODE[33640] := 16#E0F5;
   // GBK_TO_UNICODE[33641] := 16#570A;
   // GBK_TO_UNICODE[33642] := 16#E0F6;
   // GBK_TO_UNICODE[33643] := 16#5709;
   // GBK_TO_UNICODE[33644] := 16#E0F7;
   // GBK_TO_UNICODE[33645] := 16#571C;
   // GBK_TO_UNICODE[33646] := 16#E0F8;
   // GBK_TO_UNICODE[33647] := 16#5E0F;
   // GBK_TO_UNICODE[33648] := 16#E0F9;
   // GBK_TO_UNICODE[33649] := 16#5E19;
   // GBK_TO_UNICODE[33650] := 16#E0FA;
   // GBK_TO_UNICODE[33651] := 16#5E14;
   // GBK_TO_UNICODE[33652] := 16#E0FB;
   // GBK_TO_UNICODE[33653] := 16#5E11;
   // GBK_TO_UNICODE[33654] := 16#E0FC;
   // GBK_TO_UNICODE[33655] := 16#5E31;
   // GBK_TO_UNICODE[33656] := 16#E0FD;
   // GBK_TO_UNICODE[33657] := 16#5E3B;
   // GBK_TO_UNICODE[33658] := 16#E0FE;
   // GBK_TO_UNICODE[33659] := 16#5E3C;
   // GBK_TO_UNICODE[33660] := 16#E140;
   // GBK_TO_UNICODE[33661] := 16#9145;
   // GBK_TO_UNICODE[33662] := 16#E141;
   // GBK_TO_UNICODE[33663] := 16#9147;
   // GBK_TO_UNICODE[33664] := 16#E142;
   // GBK_TO_UNICODE[33665] := 16#9148;
   // GBK_TO_UNICODE[33666] := 16#E143;
   // GBK_TO_UNICODE[33667] := 16#9151;
   // GBK_TO_UNICODE[33668] := 16#E144;
   // GBK_TO_UNICODE[33669] := 16#9153;
   // GBK_TO_UNICODE[33670] := 16#E145;
   // GBK_TO_UNICODE[33671] := 16#9154;
   // GBK_TO_UNICODE[33672] := 16#E146;
   // GBK_TO_UNICODE[33673] := 16#9155;
   // GBK_TO_UNICODE[33674] := 16#E147;
   // GBK_TO_UNICODE[33675] := 16#9156;
   // GBK_TO_UNICODE[33676] := 16#E148;
   // GBK_TO_UNICODE[33677] := 16#9158;
   // GBK_TO_UNICODE[33678] := 16#E149;
   // GBK_TO_UNICODE[33679] := 16#9159;
   // GBK_TO_UNICODE[33680] := 16#E14A;
   // GBK_TO_UNICODE[33681] := 16#915B;
   // GBK_TO_UNICODE[33682] := 16#E14B;
   // GBK_TO_UNICODE[33683] := 16#915C;
   // GBK_TO_UNICODE[33684] := 16#E14C;
   // GBK_TO_UNICODE[33685] := 16#915F;
   // GBK_TO_UNICODE[33686] := 16#E14D;
   // GBK_TO_UNICODE[33687] := 16#9160;
   // GBK_TO_UNICODE[33688] := 16#E14E;
   // GBK_TO_UNICODE[33689] := 16#9166;
   // GBK_TO_UNICODE[33690] := 16#E14F;
   // GBK_TO_UNICODE[33691] := 16#9167;
   // GBK_TO_UNICODE[33692] := 16#E150;
   // GBK_TO_UNICODE[33693] := 16#9168;
   // GBK_TO_UNICODE[33694] := 16#E151;
   // GBK_TO_UNICODE[33695] := 16#916B;
   // GBK_TO_UNICODE[33696] := 16#E152;
   // GBK_TO_UNICODE[33697] := 16#916D;
   // GBK_TO_UNICODE[33698] := 16#E153;
   // GBK_TO_UNICODE[33699] := 16#9173;
   // GBK_TO_UNICODE[33700] := 16#E154;
   // GBK_TO_UNICODE[33701] := 16#917A;
   // GBK_TO_UNICODE[33702] := 16#E155;
   // GBK_TO_UNICODE[33703] := 16#917B;
   // GBK_TO_UNICODE[33704] := 16#E156;
   // GBK_TO_UNICODE[33705] := 16#917C;
   // GBK_TO_UNICODE[33706] := 16#E157;
   // GBK_TO_UNICODE[33707] := 16#9180;
   // GBK_TO_UNICODE[33708] := 16#E158;
   // GBK_TO_UNICODE[33709] := 16#9181;
   // GBK_TO_UNICODE[33710] := 16#E159;
   // GBK_TO_UNICODE[33711] := 16#9182;
   // GBK_TO_UNICODE[33712] := 16#E15A;
   // GBK_TO_UNICODE[33713] := 16#9183;
   // GBK_TO_UNICODE[33714] := 16#E15B;
   // GBK_TO_UNICODE[33715] := 16#9184;
   // GBK_TO_UNICODE[33716] := 16#E15C;
   // GBK_TO_UNICODE[33717] := 16#9186;
   // GBK_TO_UNICODE[33718] := 16#E15D;
   // GBK_TO_UNICODE[33719] := 16#9188;
   // GBK_TO_UNICODE[33720] := 16#E15E;
   // GBK_TO_UNICODE[33721] := 16#918A;
   // GBK_TO_UNICODE[33722] := 16#E15F;
   // GBK_TO_UNICODE[33723] := 16#918E;
   // GBK_TO_UNICODE[33724] := 16#E160;
   // GBK_TO_UNICODE[33725] := 16#918F;
   // GBK_TO_UNICODE[33726] := 16#E161;
   // GBK_TO_UNICODE[33727] := 16#9193;
   // GBK_TO_UNICODE[33728] := 16#E162;
   // GBK_TO_UNICODE[33729] := 16#9194;
   // GBK_TO_UNICODE[33730] := 16#E163;
   // GBK_TO_UNICODE[33731] := 16#9195;
   // GBK_TO_UNICODE[33732] := 16#E164;
   // GBK_TO_UNICODE[33733] := 16#9196;
   // GBK_TO_UNICODE[33734] := 16#E165;
   // GBK_TO_UNICODE[33735] := 16#9197;
   // GBK_TO_UNICODE[33736] := 16#E166;
   // GBK_TO_UNICODE[33737] := 16#9198;
   // GBK_TO_UNICODE[33738] := 16#E167;
   // GBK_TO_UNICODE[33739] := 16#9199;
   // GBK_TO_UNICODE[33740] := 16#E168;
   // GBK_TO_UNICODE[33741] := 16#919C;
   // GBK_TO_UNICODE[33742] := 16#E169;
   // GBK_TO_UNICODE[33743] := 16#919D;
   // GBK_TO_UNICODE[33744] := 16#E16A;
   // GBK_TO_UNICODE[33745] := 16#919E;
   // GBK_TO_UNICODE[33746] := 16#E16B;
   // GBK_TO_UNICODE[33747] := 16#919F;
   // GBK_TO_UNICODE[33748] := 16#E16C;
   // GBK_TO_UNICODE[33749] := 16#91A0;
   // GBK_TO_UNICODE[33750] := 16#E16D;
   // GBK_TO_UNICODE[33751] := 16#91A1;
   // GBK_TO_UNICODE[33752] := 16#E16E;
   // GBK_TO_UNICODE[33753] := 16#91A4;
   // GBK_TO_UNICODE[33754] := 16#E16F;
   // GBK_TO_UNICODE[33755] := 16#91A5;
   // GBK_TO_UNICODE[33756] := 16#E170;
   // GBK_TO_UNICODE[33757] := 16#91A6;
   // GBK_TO_UNICODE[33758] := 16#E171;
   // GBK_TO_UNICODE[33759] := 16#91A7;
   // GBK_TO_UNICODE[33760] := 16#E172;
   // GBK_TO_UNICODE[33761] := 16#91A8;
   // GBK_TO_UNICODE[33762] := 16#E173;
   // GBK_TO_UNICODE[33763] := 16#91A9;
   // GBK_TO_UNICODE[33764] := 16#E174;
   // GBK_TO_UNICODE[33765] := 16#91AB;
   // GBK_TO_UNICODE[33766] := 16#E175;
   // GBK_TO_UNICODE[33767] := 16#91AC;
   // GBK_TO_UNICODE[33768] := 16#E176;
   // GBK_TO_UNICODE[33769] := 16#91B0;
   // GBK_TO_UNICODE[33770] := 16#E177;
   // GBK_TO_UNICODE[33771] := 16#91B1;
   // GBK_TO_UNICODE[33772] := 16#E178;
   // GBK_TO_UNICODE[33773] := 16#91B2;
   // GBK_TO_UNICODE[33774] := 16#E179;
   // GBK_TO_UNICODE[33775] := 16#91B3;
   // GBK_TO_UNICODE[33776] := 16#E17A;
   // GBK_TO_UNICODE[33777] := 16#91B6;
   // GBK_TO_UNICODE[33778] := 16#E17B;
   // GBK_TO_UNICODE[33779] := 16#91B7;
   // GBK_TO_UNICODE[33780] := 16#E17C;
   // GBK_TO_UNICODE[33781] := 16#91B8;
   // GBK_TO_UNICODE[33782] := 16#E17D;
   // GBK_TO_UNICODE[33783] := 16#91B9;
   // GBK_TO_UNICODE[33784] := 16#E17E;
   // GBK_TO_UNICODE[33785] := 16#91BB;
   // GBK_TO_UNICODE[33786] := 16#E180;
   // GBK_TO_UNICODE[33787] := 16#91BC;
   // GBK_TO_UNICODE[33788] := 16#E181;
   // GBK_TO_UNICODE[33789] := 16#91BD;
   // GBK_TO_UNICODE[33790] := 16#E182;
   // GBK_TO_UNICODE[33791] := 16#91BE;
   // GBK_TO_UNICODE[33792] := 16#E183;
   // GBK_TO_UNICODE[33793] := 16#91BF;
   // GBK_TO_UNICODE[33794] := 16#E184;
   // GBK_TO_UNICODE[33795] := 16#91C0;
   // GBK_TO_UNICODE[33796] := 16#E185;
   // GBK_TO_UNICODE[33797] := 16#91C1;
   // GBK_TO_UNICODE[33798] := 16#E186;
   // GBK_TO_UNICODE[33799] := 16#91C2;
   // GBK_TO_UNICODE[33800] := 16#E187;
   // GBK_TO_UNICODE[33801] := 16#91C3;
   // GBK_TO_UNICODE[33802] := 16#E188;
   // GBK_TO_UNICODE[33803] := 16#91C4;
   // GBK_TO_UNICODE[33804] := 16#E189;
   // GBK_TO_UNICODE[33805] := 16#91C5;
   // GBK_TO_UNICODE[33806] := 16#E18A;
   // GBK_TO_UNICODE[33807] := 16#91C6;
   // GBK_TO_UNICODE[33808] := 16#E18B;
   // GBK_TO_UNICODE[33809] := 16#91C8;
   // GBK_TO_UNICODE[33810] := 16#E18C;
   // GBK_TO_UNICODE[33811] := 16#91CB;
   // GBK_TO_UNICODE[33812] := 16#E18D;
   // GBK_TO_UNICODE[33813] := 16#91D0;
   // GBK_TO_UNICODE[33814] := 16#E18E;
   // GBK_TO_UNICODE[33815] := 16#91D2;
   // GBK_TO_UNICODE[33816] := 16#E18F;
   // GBK_TO_UNICODE[33817] := 16#91D3;
   // GBK_TO_UNICODE[33818] := 16#E190;
   // GBK_TO_UNICODE[33819] := 16#91D4;
   // GBK_TO_UNICODE[33820] := 16#E191;
   // GBK_TO_UNICODE[33821] := 16#91D5;
   // GBK_TO_UNICODE[33822] := 16#E192;
   // GBK_TO_UNICODE[33823] := 16#91D6;
   // GBK_TO_UNICODE[33824] := 16#E193;
   // GBK_TO_UNICODE[33825] := 16#91D7;
   // GBK_TO_UNICODE[33826] := 16#E194;
   // GBK_TO_UNICODE[33827] := 16#91D8;
   // GBK_TO_UNICODE[33828] := 16#E195;
   // GBK_TO_UNICODE[33829] := 16#91D9;
   // GBK_TO_UNICODE[33830] := 16#E196;
   // GBK_TO_UNICODE[33831] := 16#91DA;
   // GBK_TO_UNICODE[33832] := 16#E197;
   // GBK_TO_UNICODE[33833] := 16#91DB;
   // GBK_TO_UNICODE[33834] := 16#E198;
   // GBK_TO_UNICODE[33835] := 16#91DD;
   // GBK_TO_UNICODE[33836] := 16#E199;
   // GBK_TO_UNICODE[33837] := 16#91DE;
   // GBK_TO_UNICODE[33838] := 16#E19A;
   // GBK_TO_UNICODE[33839] := 16#91DF;
   // GBK_TO_UNICODE[33840] := 16#E19B;
   // GBK_TO_UNICODE[33841] := 16#91E0;
   // GBK_TO_UNICODE[33842] := 16#E19C;
   // GBK_TO_UNICODE[33843] := 16#91E1;
   // GBK_TO_UNICODE[33844] := 16#E19D;
   // GBK_TO_UNICODE[33845] := 16#91E2;
   // GBK_TO_UNICODE[33846] := 16#E19E;
   // GBK_TO_UNICODE[33847] := 16#91E3;
   // GBK_TO_UNICODE[33848] := 16#E19F;
   // GBK_TO_UNICODE[33849] := 16#91E4;
   // GBK_TO_UNICODE[33850] := 16#E1A0;
   // GBK_TO_UNICODE[33851] := 16#91E5;
   // GBK_TO_UNICODE[33852] := 16#E1A1;
   // GBK_TO_UNICODE[33853] := 16#5E37;
   // GBK_TO_UNICODE[33854] := 16#E1A2;
   // GBK_TO_UNICODE[33855] := 16#5E44;
   // GBK_TO_UNICODE[33856] := 16#E1A3;
   // GBK_TO_UNICODE[33857] := 16#5E54;
   // GBK_TO_UNICODE[33858] := 16#E1A4;
   // GBK_TO_UNICODE[33859] := 16#5E5B;
   // GBK_TO_UNICODE[33860] := 16#E1A5;
   // GBK_TO_UNICODE[33861] := 16#5E5E;
   // GBK_TO_UNICODE[33862] := 16#E1A6;
   // GBK_TO_UNICODE[33863] := 16#5E61;
   // GBK_TO_UNICODE[33864] := 16#E1A7;
   // GBK_TO_UNICODE[33865] := 16#5C8C;
   // GBK_TO_UNICODE[33866] := 16#E1A8;
   // GBK_TO_UNICODE[33867] := 16#5C7A;
   // GBK_TO_UNICODE[33868] := 16#E1A9;
   // GBK_TO_UNICODE[33869] := 16#5C8D;
   // GBK_TO_UNICODE[33870] := 16#E1AA;
   // GBK_TO_UNICODE[33871] := 16#5C90;
   // GBK_TO_UNICODE[33872] := 16#E1AB;
   // GBK_TO_UNICODE[33873] := 16#5C96;
   // GBK_TO_UNICODE[33874] := 16#E1AC;
   // GBK_TO_UNICODE[33875] := 16#5C88;
   // GBK_TO_UNICODE[33876] := 16#E1AD;
   // GBK_TO_UNICODE[33877] := 16#5C98;
   // GBK_TO_UNICODE[33878] := 16#E1AE;
   // GBK_TO_UNICODE[33879] := 16#5C99;
   // GBK_TO_UNICODE[33880] := 16#E1AF;
   // GBK_TO_UNICODE[33881] := 16#5C91;
   // GBK_TO_UNICODE[33882] := 16#E1B0;
   // GBK_TO_UNICODE[33883] := 16#5C9A;
   // GBK_TO_UNICODE[33884] := 16#E1B1;
   // GBK_TO_UNICODE[33885] := 16#5C9C;
   // GBK_TO_UNICODE[33886] := 16#E1B2;
   // GBK_TO_UNICODE[33887] := 16#5CB5;
   // GBK_TO_UNICODE[33888] := 16#E1B3;
   // GBK_TO_UNICODE[33889] := 16#5CA2;
   // GBK_TO_UNICODE[33890] := 16#E1B4;
   // GBK_TO_UNICODE[33891] := 16#5CBD;
   // GBK_TO_UNICODE[33892] := 16#E1B5;
   // GBK_TO_UNICODE[33893] := 16#5CAC;
   // GBK_TO_UNICODE[33894] := 16#E1B6;
   // GBK_TO_UNICODE[33895] := 16#5CAB;
   // GBK_TO_UNICODE[33896] := 16#E1B7;
   // GBK_TO_UNICODE[33897] := 16#5CB1;
   // GBK_TO_UNICODE[33898] := 16#E1B8;
   // GBK_TO_UNICODE[33899] := 16#5CA3;
   // GBK_TO_UNICODE[33900] := 16#E1B9;
   // GBK_TO_UNICODE[33901] := 16#5CC1;
   // GBK_TO_UNICODE[33902] := 16#E1BA;
   // GBK_TO_UNICODE[33903] := 16#5CB7;
   // GBK_TO_UNICODE[33904] := 16#E1BB;
   // GBK_TO_UNICODE[33905] := 16#5CC4;
   // GBK_TO_UNICODE[33906] := 16#E1BC;
   // GBK_TO_UNICODE[33907] := 16#5CD2;
   // GBK_TO_UNICODE[33908] := 16#E1BD;
   // GBK_TO_UNICODE[33909] := 16#5CE4;
   // GBK_TO_UNICODE[33910] := 16#E1BE;
   // GBK_TO_UNICODE[33911] := 16#5CCB;
   // GBK_TO_UNICODE[33912] := 16#E1BF;
   // GBK_TO_UNICODE[33913] := 16#5CE5;
   // GBK_TO_UNICODE[33914] := 16#E1C0;
   // GBK_TO_UNICODE[33915] := 16#5D02;
   // GBK_TO_UNICODE[33916] := 16#E1C1;
   // GBK_TO_UNICODE[33917] := 16#5D03;
   // GBK_TO_UNICODE[33918] := 16#E1C2;
   // GBK_TO_UNICODE[33919] := 16#5D27;
   // GBK_TO_UNICODE[33920] := 16#E1C3;
   // GBK_TO_UNICODE[33921] := 16#5D26;
   // GBK_TO_UNICODE[33922] := 16#E1C4;
   // GBK_TO_UNICODE[33923] := 16#5D2E;
   // GBK_TO_UNICODE[33924] := 16#E1C5;
   // GBK_TO_UNICODE[33925] := 16#5D24;
   // GBK_TO_UNICODE[33926] := 16#E1C6;
   // GBK_TO_UNICODE[33927] := 16#5D1E;
   // GBK_TO_UNICODE[33928] := 16#E1C7;
   // GBK_TO_UNICODE[33929] := 16#5D06;
   // GBK_TO_UNICODE[33930] := 16#E1C8;
   // GBK_TO_UNICODE[33931] := 16#5D1B;
   // GBK_TO_UNICODE[33932] := 16#E1C9;
   // GBK_TO_UNICODE[33933] := 16#5D58;
   // GBK_TO_UNICODE[33934] := 16#E1CA;
   // GBK_TO_UNICODE[33935] := 16#5D3E;
   // GBK_TO_UNICODE[33936] := 16#E1CB;
   // GBK_TO_UNICODE[33937] := 16#5D34;
   // GBK_TO_UNICODE[33938] := 16#E1CC;
   // GBK_TO_UNICODE[33939] := 16#5D3D;
   // GBK_TO_UNICODE[33940] := 16#E1CD;
   // GBK_TO_UNICODE[33941] := 16#5D6C;
   // GBK_TO_UNICODE[33942] := 16#E1CE;
   // GBK_TO_UNICODE[33943] := 16#5D5B;
   // GBK_TO_UNICODE[33944] := 16#E1CF;
   // GBK_TO_UNICODE[33945] := 16#5D6F;
   // GBK_TO_UNICODE[33946] := 16#E1D0;
   // GBK_TO_UNICODE[33947] := 16#5D5D;
   // GBK_TO_UNICODE[33948] := 16#E1D1;
   // GBK_TO_UNICODE[33949] := 16#5D6B;
   // GBK_TO_UNICODE[33950] := 16#E1D2;
   // GBK_TO_UNICODE[33951] := 16#5D4B;
   // GBK_TO_UNICODE[33952] := 16#E1D3;
   // GBK_TO_UNICODE[33953] := 16#5D4A;
   // GBK_TO_UNICODE[33954] := 16#E1D4;
   // GBK_TO_UNICODE[33955] := 16#5D69;
   // GBK_TO_UNICODE[33956] := 16#E1D5;
   // GBK_TO_UNICODE[33957] := 16#5D74;
   // GBK_TO_UNICODE[33958] := 16#E1D6;
   // GBK_TO_UNICODE[33959] := 16#5D82;
   // GBK_TO_UNICODE[33960] := 16#E1D7;
   // GBK_TO_UNICODE[33961] := 16#5D99;
   // GBK_TO_UNICODE[33962] := 16#E1D8;
   // GBK_TO_UNICODE[33963] := 16#5D9D;
   // GBK_TO_UNICODE[33964] := 16#E1D9;
   // GBK_TO_UNICODE[33965] := 16#8C73;
   // GBK_TO_UNICODE[33966] := 16#E1DA;
   // GBK_TO_UNICODE[33967] := 16#5DB7;
   // GBK_TO_UNICODE[33968] := 16#E1DB;
   // GBK_TO_UNICODE[33969] := 16#5DC5;
   // GBK_TO_UNICODE[33970] := 16#E1DC;
   // GBK_TO_UNICODE[33971] := 16#5F73;
   // GBK_TO_UNICODE[33972] := 16#E1DD;
   // GBK_TO_UNICODE[33973] := 16#5F77;
   // GBK_TO_UNICODE[33974] := 16#E1DE;
   // GBK_TO_UNICODE[33975] := 16#5F82;
   // GBK_TO_UNICODE[33976] := 16#E1DF;
   // GBK_TO_UNICODE[33977] := 16#5F87;
   // GBK_TO_UNICODE[33978] := 16#E1E0;
   // GBK_TO_UNICODE[33979] := 16#5F89;
   // GBK_TO_UNICODE[33980] := 16#E1E1;
   // GBK_TO_UNICODE[33981] := 16#5F8C;
   // GBK_TO_UNICODE[33982] := 16#E1E2;
   // GBK_TO_UNICODE[33983] := 16#5F95;
   // GBK_TO_UNICODE[33984] := 16#E1E3;
   // GBK_TO_UNICODE[33985] := 16#5F99;
   // GBK_TO_UNICODE[33986] := 16#E1E4;
   // GBK_TO_UNICODE[33987] := 16#5F9C;
   // GBK_TO_UNICODE[33988] := 16#E1E5;
   // GBK_TO_UNICODE[33989] := 16#5FA8;
   // GBK_TO_UNICODE[33990] := 16#E1E6;
   // GBK_TO_UNICODE[33991] := 16#5FAD;
   // GBK_TO_UNICODE[33992] := 16#E1E7;
   // GBK_TO_UNICODE[33993] := 16#5FB5;
   // GBK_TO_UNICODE[33994] := 16#E1E8;
   // GBK_TO_UNICODE[33995] := 16#5FBC;
   // GBK_TO_UNICODE[33996] := 16#E1E9;
   // GBK_TO_UNICODE[33997] := 16#8862;
   // GBK_TO_UNICODE[33998] := 16#E1EA;
   // GBK_TO_UNICODE[33999] := 16#5F61;
   // GBK_TO_UNICODE[34000] := 16#E1EB;
   // GBK_TO_UNICODE[34001] := 16#72AD;
   // GBK_TO_UNICODE[34002] := 16#E1EC;
   // GBK_TO_UNICODE[34003] := 16#72B0;
   // GBK_TO_UNICODE[34004] := 16#E1ED;
   // GBK_TO_UNICODE[34005] := 16#72B4;
   // GBK_TO_UNICODE[34006] := 16#E1EE;
   // GBK_TO_UNICODE[34007] := 16#72B7;
   // GBK_TO_UNICODE[34008] := 16#E1EF;
   // GBK_TO_UNICODE[34009] := 16#72B8;
   // GBK_TO_UNICODE[34010] := 16#E1F0;
   // GBK_TO_UNICODE[34011] := 16#72C3;
   // GBK_TO_UNICODE[34012] := 16#E1F1;
   // GBK_TO_UNICODE[34013] := 16#72C1;
   // GBK_TO_UNICODE[34014] := 16#E1F2;
   // GBK_TO_UNICODE[34015] := 16#72CE;
   // GBK_TO_UNICODE[34016] := 16#E1F3;
   // GBK_TO_UNICODE[34017] := 16#72CD;
   // GBK_TO_UNICODE[34018] := 16#E1F4;
   // GBK_TO_UNICODE[34019] := 16#72D2;
   // GBK_TO_UNICODE[34020] := 16#E1F5;
   // GBK_TO_UNICODE[34021] := 16#72E8;
   // GBK_TO_UNICODE[34022] := 16#E1F6;
   // GBK_TO_UNICODE[34023] := 16#72EF;
   // GBK_TO_UNICODE[34024] := 16#E1F7;
   // GBK_TO_UNICODE[34025] := 16#72E9;
   // GBK_TO_UNICODE[34026] := 16#E1F8;
   // GBK_TO_UNICODE[34027] := 16#72F2;
   // GBK_TO_UNICODE[34028] := 16#E1F9;
   // GBK_TO_UNICODE[34029] := 16#72F4;
   // GBK_TO_UNICODE[34030] := 16#E1FA;
   // GBK_TO_UNICODE[34031] := 16#72F7;
   // GBK_TO_UNICODE[34032] := 16#E1FB;
   // GBK_TO_UNICODE[34033] := 16#7301;
   // GBK_TO_UNICODE[34034] := 16#E1FC;
   // GBK_TO_UNICODE[34035] := 16#72F3;
   // GBK_TO_UNICODE[34036] := 16#E1FD;
   // GBK_TO_UNICODE[34037] := 16#7303;
   // GBK_TO_UNICODE[34038] := 16#E1FE;
   // GBK_TO_UNICODE[34039] := 16#72FA;
   // GBK_TO_UNICODE[34040] := 16#E240;
   // GBK_TO_UNICODE[34041] := 16#91E6;
   // GBK_TO_UNICODE[34042] := 16#E241;
   // GBK_TO_UNICODE[34043] := 16#91E7;
   // GBK_TO_UNICODE[34044] := 16#E242;
   // GBK_TO_UNICODE[34045] := 16#91E8;
   // GBK_TO_UNICODE[34046] := 16#E243;
   // GBK_TO_UNICODE[34047] := 16#91E9;
   // GBK_TO_UNICODE[34048] := 16#E244;
   // GBK_TO_UNICODE[34049] := 16#91EA;
   // GBK_TO_UNICODE[34050] := 16#E245;
   // GBK_TO_UNICODE[34051] := 16#91EB;
   // GBK_TO_UNICODE[34052] := 16#E246;
   // GBK_TO_UNICODE[34053] := 16#91EC;
   // GBK_TO_UNICODE[34054] := 16#E247;
   // GBK_TO_UNICODE[34055] := 16#91ED;
   // GBK_TO_UNICODE[34056] := 16#E248;
   // GBK_TO_UNICODE[34057] := 16#91EE;
   // GBK_TO_UNICODE[34058] := 16#E249;
   // GBK_TO_UNICODE[34059] := 16#91EF;
   // GBK_TO_UNICODE[34060] := 16#E24A;
   // GBK_TO_UNICODE[34061] := 16#91F0;
   // GBK_TO_UNICODE[34062] := 16#E24B;
   // GBK_TO_UNICODE[34063] := 16#91F1;
   // GBK_TO_UNICODE[34064] := 16#E24C;
   // GBK_TO_UNICODE[34065] := 16#91F2;
   // GBK_TO_UNICODE[34066] := 16#E24D;
   // GBK_TO_UNICODE[34067] := 16#91F3;
   // GBK_TO_UNICODE[34068] := 16#E24E;
   // GBK_TO_UNICODE[34069] := 16#91F4;
   // GBK_TO_UNICODE[34070] := 16#E24F;
   // GBK_TO_UNICODE[34071] := 16#91F5;
   // GBK_TO_UNICODE[34072] := 16#E250;
   // GBK_TO_UNICODE[34073] := 16#91F6;
   // GBK_TO_UNICODE[34074] := 16#E251;
   // GBK_TO_UNICODE[34075] := 16#91F7;
   // GBK_TO_UNICODE[34076] := 16#E252;
   // GBK_TO_UNICODE[34077] := 16#91F8;
   // GBK_TO_UNICODE[34078] := 16#E253;
   // GBK_TO_UNICODE[34079] := 16#91F9;
   // GBK_TO_UNICODE[34080] := 16#E254;
   // GBK_TO_UNICODE[34081] := 16#91FA;
   // GBK_TO_UNICODE[34082] := 16#E255;
   // GBK_TO_UNICODE[34083] := 16#91FB;
   // GBK_TO_UNICODE[34084] := 16#E256;
   // GBK_TO_UNICODE[34085] := 16#91FC;
   // GBK_TO_UNICODE[34086] := 16#E257;
   // GBK_TO_UNICODE[34087] := 16#91FD;
   // GBK_TO_UNICODE[34088] := 16#E258;
   // GBK_TO_UNICODE[34089] := 16#91FE;
   // GBK_TO_UNICODE[34090] := 16#E259;
   // GBK_TO_UNICODE[34091] := 16#91FF;
   // GBK_TO_UNICODE[34092] := 16#E25A;
   // GBK_TO_UNICODE[34093] := 16#9200;
   // GBK_TO_UNICODE[34094] := 16#E25B;
   // GBK_TO_UNICODE[34095] := 16#9201;
   // GBK_TO_UNICODE[34096] := 16#E25C;
   // GBK_TO_UNICODE[34097] := 16#9202;
   // GBK_TO_UNICODE[34098] := 16#E25D;
   // GBK_TO_UNICODE[34099] := 16#9203;
   // GBK_TO_UNICODE[34100] := 16#E25E;
   // GBK_TO_UNICODE[34101] := 16#9204;
   // GBK_TO_UNICODE[34102] := 16#E25F;
   // GBK_TO_UNICODE[34103] := 16#9205;
   // GBK_TO_UNICODE[34104] := 16#E260;
   // GBK_TO_UNICODE[34105] := 16#9206;
   // GBK_TO_UNICODE[34106] := 16#E261;
   // GBK_TO_UNICODE[34107] := 16#9207;
   // GBK_TO_UNICODE[34108] := 16#E262;
   // GBK_TO_UNICODE[34109] := 16#9208;
   // GBK_TO_UNICODE[34110] := 16#E263;
   // GBK_TO_UNICODE[34111] := 16#9209;
   // GBK_TO_UNICODE[34112] := 16#E264;
   // GBK_TO_UNICODE[34113] := 16#920A;
   // GBK_TO_UNICODE[34114] := 16#E265;
   // GBK_TO_UNICODE[34115] := 16#920B;
   // GBK_TO_UNICODE[34116] := 16#E266;
   // GBK_TO_UNICODE[34117] := 16#920C;
   // GBK_TO_UNICODE[34118] := 16#E267;
   // GBK_TO_UNICODE[34119] := 16#920D;
   // GBK_TO_UNICODE[34120] := 16#E268;
   // GBK_TO_UNICODE[34121] := 16#920E;
   // GBK_TO_UNICODE[34122] := 16#E269;
   // GBK_TO_UNICODE[34123] := 16#920F;
   // GBK_TO_UNICODE[34124] := 16#E26A;
   // GBK_TO_UNICODE[34125] := 16#9210;
   // GBK_TO_UNICODE[34126] := 16#E26B;
   // GBK_TO_UNICODE[34127] := 16#9211;
   // GBK_TO_UNICODE[34128] := 16#E26C;
   // GBK_TO_UNICODE[34129] := 16#9212;
   // GBK_TO_UNICODE[34130] := 16#E26D;
   // GBK_TO_UNICODE[34131] := 16#9213;
   // GBK_TO_UNICODE[34132] := 16#E26E;
   // GBK_TO_UNICODE[34133] := 16#9214;
   // GBK_TO_UNICODE[34134] := 16#E26F;
   // GBK_TO_UNICODE[34135] := 16#9215;
   // GBK_TO_UNICODE[34136] := 16#E270;
   // GBK_TO_UNICODE[34137] := 16#9216;
   // GBK_TO_UNICODE[34138] := 16#E271;
   // GBK_TO_UNICODE[34139] := 16#9217;
   // GBK_TO_UNICODE[34140] := 16#E272;
   // GBK_TO_UNICODE[34141] := 16#9218;
   // GBK_TO_UNICODE[34142] := 16#E273;
   // GBK_TO_UNICODE[34143] := 16#9219;
   // GBK_TO_UNICODE[34144] := 16#E274;
   // GBK_TO_UNICODE[34145] := 16#921A;
   // GBK_TO_UNICODE[34146] := 16#E275;
   // GBK_TO_UNICODE[34147] := 16#921B;
   // GBK_TO_UNICODE[34148] := 16#E276;
   // GBK_TO_UNICODE[34149] := 16#921C;
   // GBK_TO_UNICODE[34150] := 16#E277;
   // GBK_TO_UNICODE[34151] := 16#921D;
   // GBK_TO_UNICODE[34152] := 16#E278;
   // GBK_TO_UNICODE[34153] := 16#921E;
   // GBK_TO_UNICODE[34154] := 16#E279;
   // GBK_TO_UNICODE[34155] := 16#921F;
   // GBK_TO_UNICODE[34156] := 16#E27A;
   // GBK_TO_UNICODE[34157] := 16#9220;
   // GBK_TO_UNICODE[34158] := 16#E27B;
   // GBK_TO_UNICODE[34159] := 16#9221;
   // GBK_TO_UNICODE[34160] := 16#E27C;
   // GBK_TO_UNICODE[34161] := 16#9222;
   // GBK_TO_UNICODE[34162] := 16#E27D;
   // GBK_TO_UNICODE[34163] := 16#9223;
   // GBK_TO_UNICODE[34164] := 16#E27E;
   // GBK_TO_UNICODE[34165] := 16#9224;
   // GBK_TO_UNICODE[34166] := 16#E280;
   // GBK_TO_UNICODE[34167] := 16#9225;
   // GBK_TO_UNICODE[34168] := 16#E281;
   // GBK_TO_UNICODE[34169] := 16#9226;
   // GBK_TO_UNICODE[34170] := 16#E282;
   // GBK_TO_UNICODE[34171] := 16#9227;
   // GBK_TO_UNICODE[34172] := 16#E283;
   // GBK_TO_UNICODE[34173] := 16#9228;
   // GBK_TO_UNICODE[34174] := 16#E284;
   // GBK_TO_UNICODE[34175] := 16#9229;
   // GBK_TO_UNICODE[34176] := 16#E285;
   // GBK_TO_UNICODE[34177] := 16#922A;
   // GBK_TO_UNICODE[34178] := 16#E286;
   // GBK_TO_UNICODE[34179] := 16#922B;
   // GBK_TO_UNICODE[34180] := 16#E287;
   // GBK_TO_UNICODE[34181] := 16#922C;
   // GBK_TO_UNICODE[34182] := 16#E288;
   // GBK_TO_UNICODE[34183] := 16#922D;
   // GBK_TO_UNICODE[34184] := 16#E289;
   // GBK_TO_UNICODE[34185] := 16#922E;
   // GBK_TO_UNICODE[34186] := 16#E28A;
   // GBK_TO_UNICODE[34187] := 16#922F;
   // GBK_TO_UNICODE[34188] := 16#E28B;
   // GBK_TO_UNICODE[34189] := 16#9230;
   // GBK_TO_UNICODE[34190] := 16#E28C;
   // GBK_TO_UNICODE[34191] := 16#9231;
   // GBK_TO_UNICODE[34192] := 16#E28D;
   // GBK_TO_UNICODE[34193] := 16#9232;
   // GBK_TO_UNICODE[34194] := 16#E28E;
   // GBK_TO_UNICODE[34195] := 16#9233;
   // GBK_TO_UNICODE[34196] := 16#E28F;
   // GBK_TO_UNICODE[34197] := 16#9234;
   // GBK_TO_UNICODE[34198] := 16#E290;
   // GBK_TO_UNICODE[34199] := 16#9235;
   // GBK_TO_UNICODE[34200] := 16#E291;
   // GBK_TO_UNICODE[34201] := 16#9236;
   // GBK_TO_UNICODE[34202] := 16#E292;
   // GBK_TO_UNICODE[34203] := 16#9237;
   // GBK_TO_UNICODE[34204] := 16#E293;
   // GBK_TO_UNICODE[34205] := 16#9238;
   // GBK_TO_UNICODE[34206] := 16#E294;
   // GBK_TO_UNICODE[34207] := 16#9239;
   // GBK_TO_UNICODE[34208] := 16#E295;
   // GBK_TO_UNICODE[34209] := 16#923A;
   // GBK_TO_UNICODE[34210] := 16#E296;
   // GBK_TO_UNICODE[34211] := 16#923B;
   // GBK_TO_UNICODE[34212] := 16#E297;
   // GBK_TO_UNICODE[34213] := 16#923C;
   // GBK_TO_UNICODE[34214] := 16#E298;
   // GBK_TO_UNICODE[34215] := 16#923D;
   // GBK_TO_UNICODE[34216] := 16#E299;
   // GBK_TO_UNICODE[34217] := 16#923E;
   // GBK_TO_UNICODE[34218] := 16#E29A;
   // GBK_TO_UNICODE[34219] := 16#923F;
   // GBK_TO_UNICODE[34220] := 16#E29B;
   // GBK_TO_UNICODE[34221] := 16#9240;
   // GBK_TO_UNICODE[34222] := 16#E29C;
   // GBK_TO_UNICODE[34223] := 16#9241;
   // GBK_TO_UNICODE[34224] := 16#E29D;
   // GBK_TO_UNICODE[34225] := 16#9242;
   // GBK_TO_UNICODE[34226] := 16#E29E;
   // GBK_TO_UNICODE[34227] := 16#9243;
   // GBK_TO_UNICODE[34228] := 16#E29F;
   // GBK_TO_UNICODE[34229] := 16#9244;
   // GBK_TO_UNICODE[34230] := 16#E2A0;
   // GBK_TO_UNICODE[34231] := 16#9245;
   // GBK_TO_UNICODE[34232] := 16#E2A1;
   // GBK_TO_UNICODE[34233] := 16#72FB;
   // GBK_TO_UNICODE[34234] := 16#E2A2;
   // GBK_TO_UNICODE[34235] := 16#7317;
   // GBK_TO_UNICODE[34236] := 16#E2A3;
   // GBK_TO_UNICODE[34237] := 16#7313;
   // GBK_TO_UNICODE[34238] := 16#E2A4;
   // GBK_TO_UNICODE[34239] := 16#7321;
   // GBK_TO_UNICODE[34240] := 16#E2A5;
   // GBK_TO_UNICODE[34241] := 16#730A;
   // GBK_TO_UNICODE[34242] := 16#E2A6;
   // GBK_TO_UNICODE[34243] := 16#731E;
   // GBK_TO_UNICODE[34244] := 16#E2A7;
   // GBK_TO_UNICODE[34245] := 16#731D;
   // GBK_TO_UNICODE[34246] := 16#E2A8;
   // GBK_TO_UNICODE[34247] := 16#7315;
   // GBK_TO_UNICODE[34248] := 16#E2A9;
   // GBK_TO_UNICODE[34249] := 16#7322;
   // GBK_TO_UNICODE[34250] := 16#E2AA;
   // GBK_TO_UNICODE[34251] := 16#7339;
   // GBK_TO_UNICODE[34252] := 16#E2AB;
   // GBK_TO_UNICODE[34253] := 16#7325;
   // GBK_TO_UNICODE[34254] := 16#E2AC;
   // GBK_TO_UNICODE[34255] := 16#732C;
   // GBK_TO_UNICODE[34256] := 16#E2AD;
   // GBK_TO_UNICODE[34257] := 16#7338;
   // GBK_TO_UNICODE[34258] := 16#E2AE;
   // GBK_TO_UNICODE[34259] := 16#7331;
   // GBK_TO_UNICODE[34260] := 16#E2AF;
   // GBK_TO_UNICODE[34261] := 16#7350;
   // GBK_TO_UNICODE[34262] := 16#E2B0;
   // GBK_TO_UNICODE[34263] := 16#734D;
   // GBK_TO_UNICODE[34264] := 16#E2B1;
   // GBK_TO_UNICODE[34265] := 16#7357;
   // GBK_TO_UNICODE[34266] := 16#E2B2;
   // GBK_TO_UNICODE[34267] := 16#7360;
   // GBK_TO_UNICODE[34268] := 16#E2B3;
   // GBK_TO_UNICODE[34269] := 16#736C;
   // GBK_TO_UNICODE[34270] := 16#E2B4;
   // GBK_TO_UNICODE[34271] := 16#736F;
   // GBK_TO_UNICODE[34272] := 16#E2B5;
   // GBK_TO_UNICODE[34273] := 16#737E;
   // GBK_TO_UNICODE[34274] := 16#E2B6;
   // GBK_TO_UNICODE[34275] := 16#821B;
   // GBK_TO_UNICODE[34276] := 16#E2B7;
   // GBK_TO_UNICODE[34277] := 16#5925;
   // GBK_TO_UNICODE[34278] := 16#E2B8;
   // GBK_TO_UNICODE[34279] := 16#98E7;
   // GBK_TO_UNICODE[34280] := 16#E2B9;
   // GBK_TO_UNICODE[34281] := 16#5924;
   // GBK_TO_UNICODE[34282] := 16#E2BA;
   // GBK_TO_UNICODE[34283] := 16#5902;
   // GBK_TO_UNICODE[34284] := 16#E2BB;
   // GBK_TO_UNICODE[34285] := 16#9963;
   // GBK_TO_UNICODE[34286] := 16#E2BC;
   // GBK_TO_UNICODE[34287] := 16#9967;
   // GBK_TO_UNICODE[34288] := 16#E2BD;
   // GBK_TO_UNICODE[34289] := 16#9968;
   // GBK_TO_UNICODE[34290] := 16#E2BE;
   // GBK_TO_UNICODE[34291] := 16#9969;
   // GBK_TO_UNICODE[34292] := 16#E2BF;
   // GBK_TO_UNICODE[34293] := 16#996A;
   // GBK_TO_UNICODE[34294] := 16#E2C0;
   // GBK_TO_UNICODE[34295] := 16#996B;
   // GBK_TO_UNICODE[34296] := 16#E2C1;
   // GBK_TO_UNICODE[34297] := 16#996C;
   // GBK_TO_UNICODE[34298] := 16#E2C2;
   // GBK_TO_UNICODE[34299] := 16#9974;
   // GBK_TO_UNICODE[34300] := 16#E2C3;
   // GBK_TO_UNICODE[34301] := 16#9977;
   // GBK_TO_UNICODE[34302] := 16#E2C4;
   // GBK_TO_UNICODE[34303] := 16#997D;
   // GBK_TO_UNICODE[34304] := 16#E2C5;
   // GBK_TO_UNICODE[34305] := 16#9980;
   // GBK_TO_UNICODE[34306] := 16#E2C6;
   // GBK_TO_UNICODE[34307] := 16#9984;
   // GBK_TO_UNICODE[34308] := 16#E2C7;
   // GBK_TO_UNICODE[34309] := 16#9987;
   // GBK_TO_UNICODE[34310] := 16#E2C8;
   // GBK_TO_UNICODE[34311] := 16#998A;
   // GBK_TO_UNICODE[34312] := 16#E2C9;
   // GBK_TO_UNICODE[34313] := 16#998D;
   // GBK_TO_UNICODE[34314] := 16#E2CA;
   // GBK_TO_UNICODE[34315] := 16#9990;
   // GBK_TO_UNICODE[34316] := 16#E2CB;
   // GBK_TO_UNICODE[34317] := 16#9991;
   // GBK_TO_UNICODE[34318] := 16#E2CC;
   // GBK_TO_UNICODE[34319] := 16#9993;
   // GBK_TO_UNICODE[34320] := 16#E2CD;
   // GBK_TO_UNICODE[34321] := 16#9994;
   // GBK_TO_UNICODE[34322] := 16#E2CE;
   // GBK_TO_UNICODE[34323] := 16#9995;
   // GBK_TO_UNICODE[34324] := 16#E2CF;
   // GBK_TO_UNICODE[34325] := 16#5E80;
   // GBK_TO_UNICODE[34326] := 16#E2D0;
   // GBK_TO_UNICODE[34327] := 16#5E91;
   // GBK_TO_UNICODE[34328] := 16#E2D1;
   // GBK_TO_UNICODE[34329] := 16#5E8B;
   // GBK_TO_UNICODE[34330] := 16#E2D2;
   // GBK_TO_UNICODE[34331] := 16#5E96;
   // GBK_TO_UNICODE[34332] := 16#E2D3;
   // GBK_TO_UNICODE[34333] := 16#5EA5;
   // GBK_TO_UNICODE[34334] := 16#E2D4;
   // GBK_TO_UNICODE[34335] := 16#5EA0;
   // GBK_TO_UNICODE[34336] := 16#E2D5;
   // GBK_TO_UNICODE[34337] := 16#5EB9;
   // GBK_TO_UNICODE[34338] := 16#E2D6;
   // GBK_TO_UNICODE[34339] := 16#5EB5;
   // GBK_TO_UNICODE[34340] := 16#E2D7;
   // GBK_TO_UNICODE[34341] := 16#5EBE;
   // GBK_TO_UNICODE[34342] := 16#E2D8;
   // GBK_TO_UNICODE[34343] := 16#5EB3;
   // GBK_TO_UNICODE[34344] := 16#E2D9;
   // GBK_TO_UNICODE[34345] := 16#8D53;
   // GBK_TO_UNICODE[34346] := 16#E2DA;
   // GBK_TO_UNICODE[34347] := 16#5ED2;
   // GBK_TO_UNICODE[34348] := 16#E2DB;
   // GBK_TO_UNICODE[34349] := 16#5ED1;
   // GBK_TO_UNICODE[34350] := 16#E2DC;
   // GBK_TO_UNICODE[34351] := 16#5EDB;
   // GBK_TO_UNICODE[34352] := 16#E2DD;
   // GBK_TO_UNICODE[34353] := 16#5EE8;
   // GBK_TO_UNICODE[34354] := 16#E2DE;
   // GBK_TO_UNICODE[34355] := 16#5EEA;
   // GBK_TO_UNICODE[34356] := 16#E2DF;
   // GBK_TO_UNICODE[34357] := 16#81BA;
   // GBK_TO_UNICODE[34358] := 16#E2E0;
   // GBK_TO_UNICODE[34359] := 16#5FC4;
   // GBK_TO_UNICODE[34360] := 16#E2E1;
   // GBK_TO_UNICODE[34361] := 16#5FC9;
   // GBK_TO_UNICODE[34362] := 16#E2E2;
   // GBK_TO_UNICODE[34363] := 16#5FD6;
   // GBK_TO_UNICODE[34364] := 16#E2E3;
   // GBK_TO_UNICODE[34365] := 16#5FCF;
   // GBK_TO_UNICODE[34366] := 16#E2E4;
   // GBK_TO_UNICODE[34367] := 16#6003;
   // GBK_TO_UNICODE[34368] := 16#E2E5;
   // GBK_TO_UNICODE[34369] := 16#5FEE;
   // GBK_TO_UNICODE[34370] := 16#E2E6;
   // GBK_TO_UNICODE[34371] := 16#6004;
   // GBK_TO_UNICODE[34372] := 16#E2E7;
   // GBK_TO_UNICODE[34373] := 16#5FE1;
   // GBK_TO_UNICODE[34374] := 16#E2E8;
   // GBK_TO_UNICODE[34375] := 16#5FE4;
   // GBK_TO_UNICODE[34376] := 16#E2E9;
   // GBK_TO_UNICODE[34377] := 16#5FFE;
   // GBK_TO_UNICODE[34378] := 16#E2EA;
   // GBK_TO_UNICODE[34379] := 16#6005;
   // GBK_TO_UNICODE[34380] := 16#E2EB;
   // GBK_TO_UNICODE[34381] := 16#6006;
   // GBK_TO_UNICODE[34382] := 16#E2EC;
   // GBK_TO_UNICODE[34383] := 16#5FEA;
   // GBK_TO_UNICODE[34384] := 16#E2ED;
   // GBK_TO_UNICODE[34385] := 16#5FED;
   // GBK_TO_UNICODE[34386] := 16#E2EE;
   // GBK_TO_UNICODE[34387] := 16#5FF8;
   // GBK_TO_UNICODE[34388] := 16#E2EF;
   // GBK_TO_UNICODE[34389] := 16#6019;
   // GBK_TO_UNICODE[34390] := 16#E2F0;
   // GBK_TO_UNICODE[34391] := 16#6035;
   // GBK_TO_UNICODE[34392] := 16#E2F1;
   // GBK_TO_UNICODE[34393] := 16#6026;
   // GBK_TO_UNICODE[34394] := 16#E2F2;
   // GBK_TO_UNICODE[34395] := 16#601B;
   // GBK_TO_UNICODE[34396] := 16#E2F3;
   // GBK_TO_UNICODE[34397] := 16#600F;
   // GBK_TO_UNICODE[34398] := 16#E2F4;
   // GBK_TO_UNICODE[34399] := 16#600D;
   // GBK_TO_UNICODE[34400] := 16#E2F5;
   // GBK_TO_UNICODE[34401] := 16#6029;
   // GBK_TO_UNICODE[34402] := 16#E2F6;
   // GBK_TO_UNICODE[34403] := 16#602B;
   // GBK_TO_UNICODE[34404] := 16#E2F7;
   // GBK_TO_UNICODE[34405] := 16#600A;
   // GBK_TO_UNICODE[34406] := 16#E2F8;
   // GBK_TO_UNICODE[34407] := 16#603F;
   // GBK_TO_UNICODE[34408] := 16#E2F9;
   // GBK_TO_UNICODE[34409] := 16#6021;
   // GBK_TO_UNICODE[34410] := 16#E2FA;
   // GBK_TO_UNICODE[34411] := 16#6078;
   // GBK_TO_UNICODE[34412] := 16#E2FB;
   // GBK_TO_UNICODE[34413] := 16#6079;
   // GBK_TO_UNICODE[34414] := 16#E2FC;
   // GBK_TO_UNICODE[34415] := 16#607B;
   // GBK_TO_UNICODE[34416] := 16#E2FD;
   // GBK_TO_UNICODE[34417] := 16#607A;
   // GBK_TO_UNICODE[34418] := 16#E2FE;
   // GBK_TO_UNICODE[34419] := 16#6042;
   // GBK_TO_UNICODE[34420] := 16#E340;
   // GBK_TO_UNICODE[34421] := 16#9246;
   // GBK_TO_UNICODE[34422] := 16#E341;
   // GBK_TO_UNICODE[34423] := 16#9247;
   // GBK_TO_UNICODE[34424] := 16#E342;
   // GBK_TO_UNICODE[34425] := 16#9248;
   // GBK_TO_UNICODE[34426] := 16#E343;
   // GBK_TO_UNICODE[34427] := 16#9249;
   // GBK_TO_UNICODE[34428] := 16#E344;
   // GBK_TO_UNICODE[34429] := 16#924A;
   // GBK_TO_UNICODE[34430] := 16#E345;
   // GBK_TO_UNICODE[34431] := 16#924B;
   // GBK_TO_UNICODE[34432] := 16#E346;
   // GBK_TO_UNICODE[34433] := 16#924C;
   // GBK_TO_UNICODE[34434] := 16#E347;
   // GBK_TO_UNICODE[34435] := 16#924D;
   // GBK_TO_UNICODE[34436] := 16#E348;
   // GBK_TO_UNICODE[34437] := 16#924E;
   // GBK_TO_UNICODE[34438] := 16#E349;
   // GBK_TO_UNICODE[34439] := 16#924F;
   // GBK_TO_UNICODE[34440] := 16#E34A;
   // GBK_TO_UNICODE[34441] := 16#9250;
   // GBK_TO_UNICODE[34442] := 16#E34B;
   // GBK_TO_UNICODE[34443] := 16#9251;
   // GBK_TO_UNICODE[34444] := 16#E34C;
   // GBK_TO_UNICODE[34445] := 16#9252;
   // GBK_TO_UNICODE[34446] := 16#E34D;
   // GBK_TO_UNICODE[34447] := 16#9253;
   // GBK_TO_UNICODE[34448] := 16#E34E;
   // GBK_TO_UNICODE[34449] := 16#9254;
   // GBK_TO_UNICODE[34450] := 16#E34F;
   // GBK_TO_UNICODE[34451] := 16#9255;
   // GBK_TO_UNICODE[34452] := 16#E350;
   // GBK_TO_UNICODE[34453] := 16#9256;
   // GBK_TO_UNICODE[34454] := 16#E351;
   // GBK_TO_UNICODE[34455] := 16#9257;
   // GBK_TO_UNICODE[34456] := 16#E352;
   // GBK_TO_UNICODE[34457] := 16#9258;
   // GBK_TO_UNICODE[34458] := 16#E353;
   // GBK_TO_UNICODE[34459] := 16#9259;
   // GBK_TO_UNICODE[34460] := 16#E354;
   // GBK_TO_UNICODE[34461] := 16#925A;
   // GBK_TO_UNICODE[34462] := 16#E355;
   // GBK_TO_UNICODE[34463] := 16#925B;
   // GBK_TO_UNICODE[34464] := 16#E356;
   // GBK_TO_UNICODE[34465] := 16#925C;
   // GBK_TO_UNICODE[34466] := 16#E357;
   // GBK_TO_UNICODE[34467] := 16#925D;
   // GBK_TO_UNICODE[34468] := 16#E358;
   // GBK_TO_UNICODE[34469] := 16#925E;
   // GBK_TO_UNICODE[34470] := 16#E359;
   // GBK_TO_UNICODE[34471] := 16#925F;
   // GBK_TO_UNICODE[34472] := 16#E35A;
   // GBK_TO_UNICODE[34473] := 16#9260;
   // GBK_TO_UNICODE[34474] := 16#E35B;
   // GBK_TO_UNICODE[34475] := 16#9261;
   // GBK_TO_UNICODE[34476] := 16#E35C;
   // GBK_TO_UNICODE[34477] := 16#9262;
   // GBK_TO_UNICODE[34478] := 16#E35D;
   // GBK_TO_UNICODE[34479] := 16#9263;
   // GBK_TO_UNICODE[34480] := 16#E35E;
   // GBK_TO_UNICODE[34481] := 16#9264;
   // GBK_TO_UNICODE[34482] := 16#E35F;
   // GBK_TO_UNICODE[34483] := 16#9265;
   // GBK_TO_UNICODE[34484] := 16#E360;
   // GBK_TO_UNICODE[34485] := 16#9266;
   // GBK_TO_UNICODE[34486] := 16#E361;
   // GBK_TO_UNICODE[34487] := 16#9267;
   // GBK_TO_UNICODE[34488] := 16#E362;
   // GBK_TO_UNICODE[34489] := 16#9268;
   // GBK_TO_UNICODE[34490] := 16#E363;
   // GBK_TO_UNICODE[34491] := 16#9269;
   // GBK_TO_UNICODE[34492] := 16#E364;
   // GBK_TO_UNICODE[34493] := 16#926A;
   // GBK_TO_UNICODE[34494] := 16#E365;
   // GBK_TO_UNICODE[34495] := 16#926B;
   // GBK_TO_UNICODE[34496] := 16#E366;
   // GBK_TO_UNICODE[34497] := 16#926C;
   // GBK_TO_UNICODE[34498] := 16#E367;
   // GBK_TO_UNICODE[34499] := 16#926D;
   // GBK_TO_UNICODE[34500] := 16#E368;
   // GBK_TO_UNICODE[34501] := 16#926E;
   // GBK_TO_UNICODE[34502] := 16#E369;
   // GBK_TO_UNICODE[34503] := 16#926F;
   // GBK_TO_UNICODE[34504] := 16#E36A;
   // GBK_TO_UNICODE[34505] := 16#9270;
   // GBK_TO_UNICODE[34506] := 16#E36B;
   // GBK_TO_UNICODE[34507] := 16#9271;
   // GBK_TO_UNICODE[34508] := 16#E36C;
   // GBK_TO_UNICODE[34509] := 16#9272;
   // GBK_TO_UNICODE[34510] := 16#E36D;
   // GBK_TO_UNICODE[34511] := 16#9273;
   // GBK_TO_UNICODE[34512] := 16#E36E;
   // GBK_TO_UNICODE[34513] := 16#9275;
   // GBK_TO_UNICODE[34514] := 16#E36F;
   // GBK_TO_UNICODE[34515] := 16#9276;
   // GBK_TO_UNICODE[34516] := 16#E370;
   // GBK_TO_UNICODE[34517] := 16#9277;
   // GBK_TO_UNICODE[34518] := 16#E371;
   // GBK_TO_UNICODE[34519] := 16#9278;
   // GBK_TO_UNICODE[34520] := 16#E372;
   // GBK_TO_UNICODE[34521] := 16#9279;
   // GBK_TO_UNICODE[34522] := 16#E373;
   // GBK_TO_UNICODE[34523] := 16#927A;
   // GBK_TO_UNICODE[34524] := 16#E374;
   // GBK_TO_UNICODE[34525] := 16#927B;
   // GBK_TO_UNICODE[34526] := 16#E375;
   // GBK_TO_UNICODE[34527] := 16#927C;
   // GBK_TO_UNICODE[34528] := 16#E376;
   // GBK_TO_UNICODE[34529] := 16#927D;
   // GBK_TO_UNICODE[34530] := 16#E377;
   // GBK_TO_UNICODE[34531] := 16#927E;
   // GBK_TO_UNICODE[34532] := 16#E378;
   // GBK_TO_UNICODE[34533] := 16#927F;
   // GBK_TO_UNICODE[34534] := 16#E379;
   // GBK_TO_UNICODE[34535] := 16#9280;
   // GBK_TO_UNICODE[34536] := 16#E37A;
   // GBK_TO_UNICODE[34537] := 16#9281;
   // GBK_TO_UNICODE[34538] := 16#E37B;
   // GBK_TO_UNICODE[34539] := 16#9282;
   // GBK_TO_UNICODE[34540] := 16#E37C;
   // GBK_TO_UNICODE[34541] := 16#9283;
   // GBK_TO_UNICODE[34542] := 16#E37D;
   // GBK_TO_UNICODE[34543] := 16#9284;
   // GBK_TO_UNICODE[34544] := 16#E37E;
   // GBK_TO_UNICODE[34545] := 16#9285;
   // GBK_TO_UNICODE[34546] := 16#E380;
   // GBK_TO_UNICODE[34547] := 16#9286;
   // GBK_TO_UNICODE[34548] := 16#E381;
   // GBK_TO_UNICODE[34549] := 16#9287;
   // GBK_TO_UNICODE[34550] := 16#E382;
   // GBK_TO_UNICODE[34551] := 16#9288;
   // GBK_TO_UNICODE[34552] := 16#E383;
   // GBK_TO_UNICODE[34553] := 16#9289;
   // GBK_TO_UNICODE[34554] := 16#E384;
   // GBK_TO_UNICODE[34555] := 16#928A;
   // GBK_TO_UNICODE[34556] := 16#E385;
   // GBK_TO_UNICODE[34557] := 16#928B;
   // GBK_TO_UNICODE[34558] := 16#E386;
   // GBK_TO_UNICODE[34559] := 16#928C;
   // GBK_TO_UNICODE[34560] := 16#E387;
   // GBK_TO_UNICODE[34561] := 16#928D;
   // GBK_TO_UNICODE[34562] := 16#E388;
   // GBK_TO_UNICODE[34563] := 16#928F;
   // GBK_TO_UNICODE[34564] := 16#E389;
   // GBK_TO_UNICODE[34565] := 16#9290;
   // GBK_TO_UNICODE[34566] := 16#E38A;
   // GBK_TO_UNICODE[34567] := 16#9291;
